// TIA Portal V17 export
// export: Created 2025-03-05T08:03:02.1046817Z, ExportSetting WithDefaults, DisplayName Totally Integrated Automation Portal, DisplayVersion V17 Update 8, DisplayName TIA Portal Openness, DisplayVersion V17 Update 8, DisplayName TIA Portal Version Control Interface, DisplayVersion V17, DisplayName SINAMICS Startdrive Advanced, DisplayVersion V17 SP2, DisplayName SINAMICS Startdrive G110M, G120, G120C, G120D, G120P, G115D, DisplayVersion V17 SP2, DisplayName SINAMICS Startdrive G130, G150, S120, S150, SINAMICS MV, S210, DisplayVersion V17 SP2, DisplayName STEP 7 Professional, DisplayVersion V17 Update 8, DisplayName SINUMERIK ONE STEP 7 Toolbox, DisplayVersion V17 Update 12, DisplayName SINUMERIK 840D sl STEP 7 Toolbox, DisplayVersion V17 Update 12, DisplayName STEP 7 Safety, DisplayVersion V17 Update 6, DisplayName WinCC Advanced, DisplayVersion V17 Update 8
FUNCTION "FC21013_POWDER_FEEDER_HOPPER" : Void   // FC21013, LAD
TITLE = FC21011 POWDER FEEDER HOPPER
{ S7_Optimized_Access := 'TRUE' }
VERSION : 0.1
// stored: AutoNumber false, IsIECCheckEnabled false, SetENOAutomatically false, UDAEnableTagReadback false
   VAR_TEMP
      AUX_PRESSURE : Int;
      AUX_DIGITAL1 : Bool;
      AUX_DIGITAL2 : Bool;
      AUX_SCATTER : Array[0..15] of Bool;
      PRESSURE_NORM : Real;
      PRESSURE_SCALE : Real;
      AUX_PRESSURE2 : Real;
      SCALED2 : Real;
   END_VAR
BEGIN

REGION Network 1: /////_UNIT_01_/////
END_REGION

REGION Network 2: CALL FB21013 POWDER FEEDER 1 HOPPER UNIT 01
   // 2#0000_0001 OPTIONS 0 BIT 0 LINE 1 ENABLED OPTION
   // 2#0000_0010 OPTIONS 0 BIT 1 LINE 2 ENABLED OPTION
   // 2#0000_0100 OPTIONS 0 BIT 2 SPARE
   // 2#0000_1000 OPTIONS 0 BIT 3 SPARE
   // 2#0001_0000 OPTIONS 0 BIT 4 SPARE
   // 2#0010_0000 OPTIONS 0 BIT 5 SPARE
   // 2#0100_0000 OPTIONS 0 BIT 6 SPARE
   // 2#1000_0000 OPTIONS 0 BIT 7 SPARE
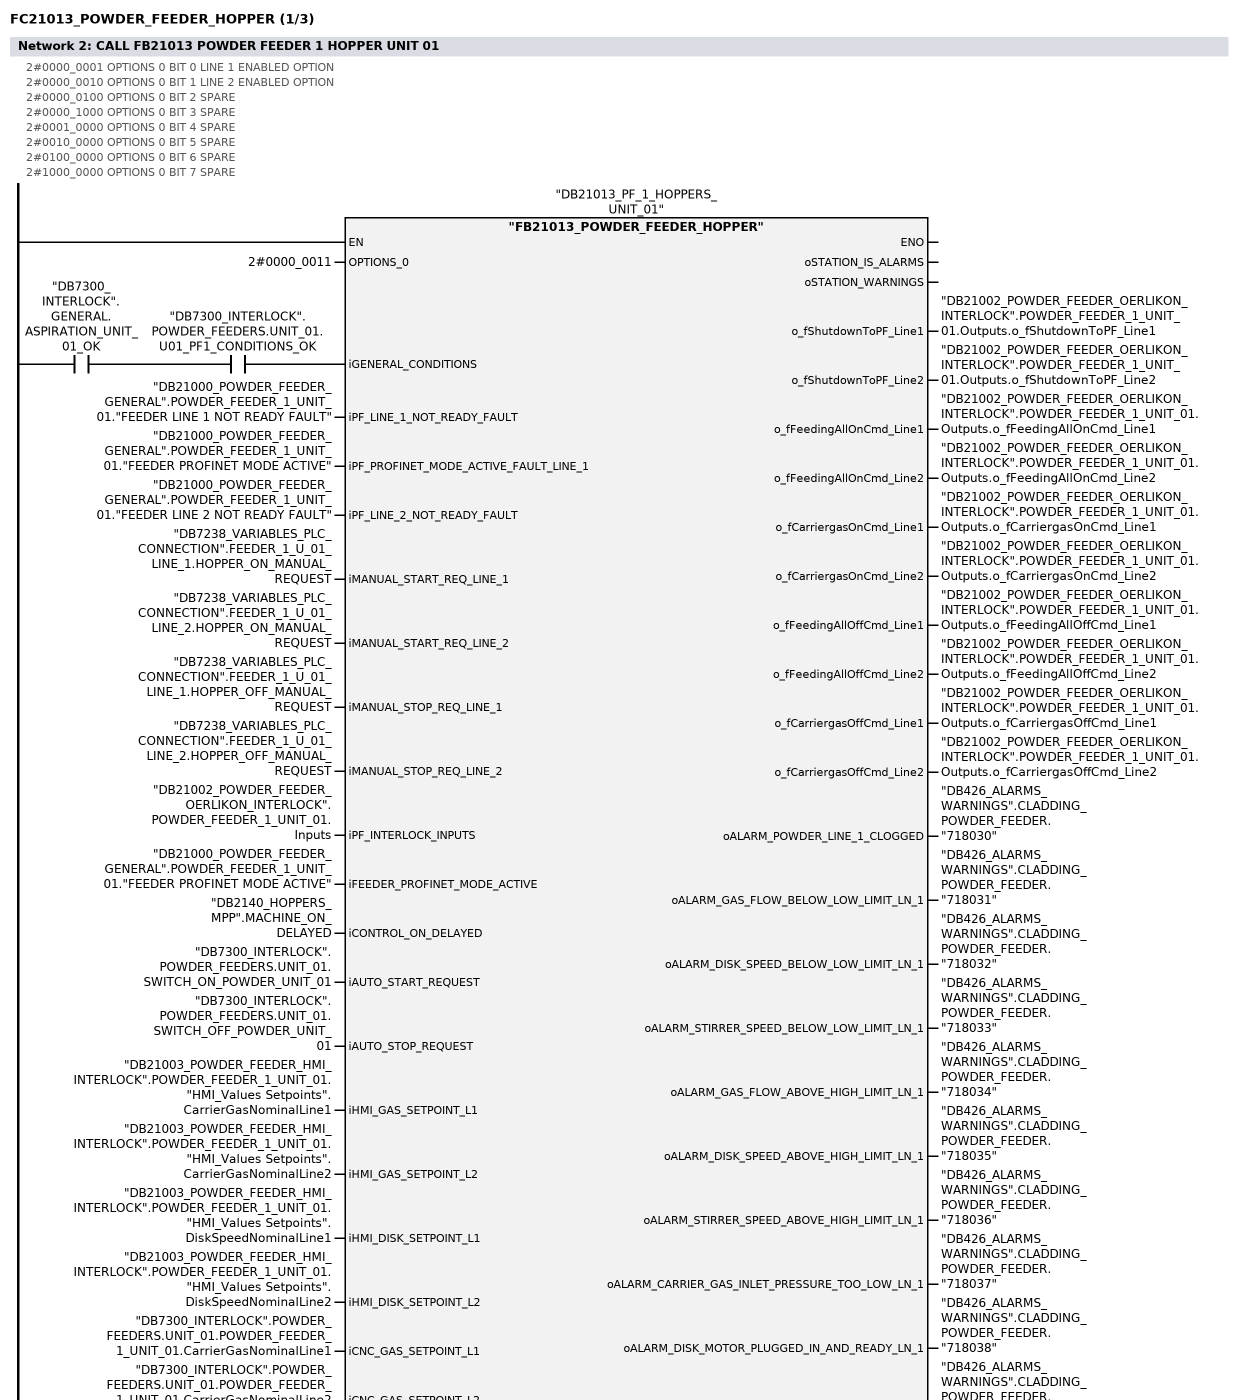
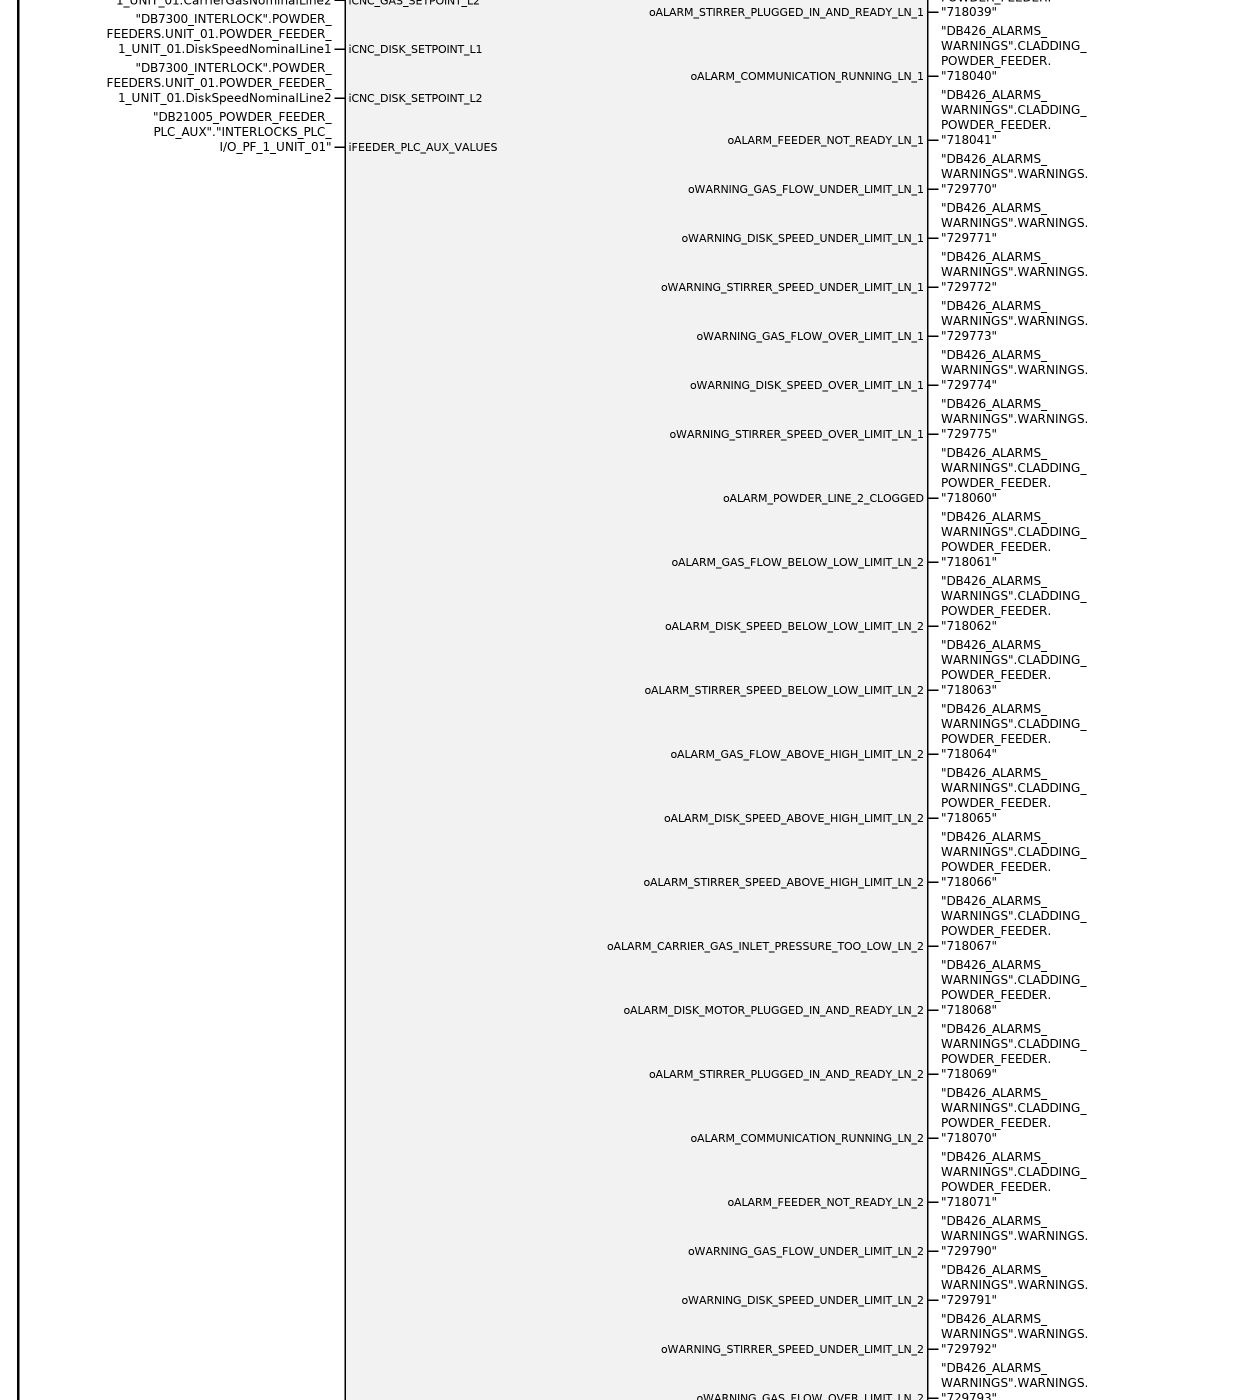
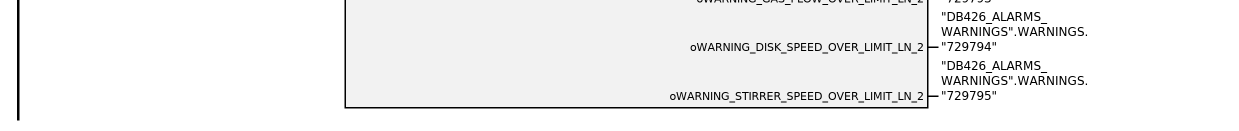
   RUNG wire#powerrail
      "DB21013_PF_1_HOPPERS_UNIT_01"(iGENERAL_CONDITIONS := wire#w1, OPTIONS_0 := 2#0000_0011, iPF_LINE_1_NOT_READY_FAULT := "DB21000_POWDER_FEEDER_GENERAL".POWDER_FEEDER_1_UNIT_01."FEEDER LINE 1 NOT READY FAULT", iPF_PROFINET_MODE_ACTIVE_FAULT_LINE_1 := "DB21000_POWDER_FEEDER_GENERAL".POWDER_FEEDER_1_UNIT_01."FEEDER PROFINET MODE ACTIVE", iPF_LINE_2_NOT_READY_FAULT := "DB21000_POWDER_FEEDER_GENERAL".POWDER_FEEDER_1_UNIT_01."FEEDER LINE 2 NOT READY FAULT", iMANUAL_START_REQ_LINE_1 := "DB7238_VARIABLES_PLC_CONNECTION".FEEDER_1_U_01_LINE_1.HOPPER_ON_MANUAL_REQUEST, iMANUAL_START_REQ_LINE_2 := "DB7238_VARIABLES_PLC_CONNECTION".FEEDER_1_U_01_LINE_2.HOPPER_ON_MANUAL_REQUEST, iMANUAL_STOP_REQ_LINE_1 := "DB7238_VARIABLES_PLC_CONNECTION".FEEDER_1_U_01_LINE_1.HOPPER_OFF_MANUAL_REQUEST, iMANUAL_STOP_REQ_LINE_2 := "DB7238_VARIABLES_PLC_CONNECTION".FEEDER_1_U_01_LINE_2.HOPPER_OFF_MANUAL_REQUEST, iPF_INTERLOCK_INPUTS := "DB21002_POWDER_FEEDER_OERLIKON_INTERLOCK".POWDER_FEEDER_1_UNIT_01.Inputs, iFEEDER_PROFINET_MODE_ACTIVE := "DB21000_POWDER_FEEDER_GENERAL".POWDER_FEEDER_1_UNIT_01."FEEDER PROFINET MODE ACTIVE", iCONTROL_ON_DELAYED := "DB2140_HOPPERS_MPP".MACHINE_ON_DELAYED, iAUTO_START_REQUEST := "DB7300_INTERLOCK".POWDER_FEEDERS.UNIT_01.SWITCH_ON_POWDER_UNIT_01, iAUTO_STOP_REQUEST := "DB7300_INTERLOCK".POWDER_FEEDERS.UNIT_01.SWITCH_OFF_POWDER_UNIT_01, iHMI_GAS_SETPOINT_L1 := "DB21003_POWDER_FEEDER_HMI_INTERLOCK".POWDER_FEEDER_1_UNIT_01."HMI_Values Setpoints".CarrierGasNominalLine1, iHMI_GAS_SETPOINT_L2 := "DB21003_POWDER_FEEDER_HMI_INTERLOCK".POWDER_FEEDER_1_UNIT_01."HMI_Values Setpoints".CarrierGasNominalLine2, iHMI_DISK_SETPOINT_L1 := "DB21003_POWDER_FEEDER_HMI_INTERLOCK".POWDER_FEEDER_1_UNIT_01."HMI_Values Setpoints".DiskSpeedNominalLine1, iHMI_DISK_SETPOINT_L2 := "DB21003_POWDER_FEEDER_HMI_INTERLOCK".POWDER_FEEDER_1_UNIT_01."HMI_Values Setpoints".DiskSpeedNominalLine2, iCNC_GAS_SETPOINT_L1 := "DB7300_INTERLOCK".POWDER_FEEDERS.UNIT_01.POWDER_FEEDER_1_UNIT_01.CarrierGasNominalLine1, iCNC_GAS_SETPOINT_L2 := "DB7300_INTERLOCK".POWDER_FEEDERS.UNIT_01.POWDER_FEEDER_1_UNIT_01.CarrierGasNominalLine2, iCNC_DISK_SETPOINT_L1 := "DB7300_INTERLOCK".POWDER_FEEDERS.UNIT_01.POWDER_FEEDER_1_UNIT_01.DiskSpeedNominalLine1, iCNC_DISK_SETPOINT_L2 := "DB7300_INTERLOCK".POWDER_FEEDERS.UNIT_01.POWDER_FEEDER_1_UNIT_01.DiskSpeedNominalLine2, iFEEDER_PLC_AUX_VALUES := "DB21005_POWDER_FEEDER_PLC_AUX"."INTERLOCKS_PLC_I/O_PF_1_UNIT_01", oSTATION_IS_ALARMS =>, oSTATION_WARNINGS =>, o_fShutdownToPF_Line1 => "DB21002_POWDER_FEEDER_OERLIKON_INTERLOCK".POWDER_FEEDER_1_UNIT_01.Outputs.o_fShutdownToPF_Line1, o_fShutdownToPF_Line2 => "DB21002_POWDER_FEEDER_OERLIKON_INTERLOCK".POWDER_FEEDER_1_UNIT_01.Outputs.o_fShutdownToPF_Line2, o_fFeedingAllOnCmd_Line1 => "DB21002_POWDER_FEEDER_OERLIKON_INTERLOCK".POWDER_FEEDER_1_UNIT_01.Outputs.o_fFeedingAllOnCmd_Line1, o_fFeedingAllOnCmd_Line2 => "DB21002_POWDER_FEEDER_OERLIKON_INTERLOCK".POWDER_FEEDER_1_UNIT_01.Outputs.o_fFeedingAllOnCmd_Line2, o_fCarriergasOnCmd_Line1 => "DB21002_POWDER_FEEDER_OERLIKON_INTERLOCK".POWDER_FEEDER_1_UNIT_01.Outputs.o_fCarriergasOnCmd_Line1, o_fCarriergasOnCmd_Line2 => "DB21002_POWDER_FEEDER_OERLIKON_INTERLOCK".POWDER_FEEDER_1_UNIT_01.Outputs.o_fCarriergasOnCmd_Line2, o_fFeedingAllOffCmd_Line1 => "DB21002_POWDER_FEEDER_OERLIKON_INTERLOCK".POWDER_FEEDER_1_UNIT_01.Outputs.o_fFeedingAllOffCmd_Line1, o_fFeedingAllOffCmd_Line2 => "DB21002_POWDER_FEEDER_OERLIKON_INTERLOCK".POWDER_FEEDER_1_UNIT_01.Outputs.o_fFeedingAllOffCmd_Line2, o_fCarriergasOffCmd_Line1 => "DB21002_POWDER_FEEDER_OERLIKON_INTERLOCK".POWDER_FEEDER_1_UNIT_01.Outputs.o_fCarriergasOffCmd_Line1, o_fCarriergasOffCmd_Line2 => "DB21002_POWDER_FEEDER_OERLIKON_INTERLOCK".POWDER_FEEDER_1_UNIT_01.Outputs.o_fCarriergasOffCmd_Line2, oALARM_POWDER_LINE_1_CLOGGED => "DB426_ALARMS_WARNINGS".CLADDING_POWDER_FEEDER."718030", oALARM_GAS_FLOW_BELOW_LOW_LIMIT_LN_1 => "DB426_ALARMS_WARNINGS".CLADDING_POWDER_FEEDER."718031", oALARM_DISK_SPEED_BELOW_LOW_LIMIT_LN_1 => "DB426_ALARMS_WARNINGS".CLADDING_POWDER_FEEDER."718032", oALARM_STIRRER_SPEED_BELOW_LOW_LIMIT_LN_1 => "DB426_ALARMS_WARNINGS".CLADDING_POWDER_FEEDER."718033", oALARM_GAS_FLOW_ABOVE_HIGH_LIMIT_LN_1 => "DB426_ALARMS_WARNINGS".CLADDING_POWDER_FEEDER."718034", oALARM_DISK_SPEED_ABOVE_HIGH_LIMIT_LN_1 => "DB426_ALARMS_WARNINGS".CLADDING_POWDER_FEEDER."718035", oALARM_STIRRER_SPEED_ABOVE_HIGH_LIMIT_LN_1 => "DB426_ALARMS_WARNINGS".CLADDING_POWDER_FEEDER."718036", oALARM_CARRIER_GAS_INLET_PRESSURE_TOO_LOW_LN_1 => "DB426_ALARMS_WARNINGS".CLADDING_POWDER_FEEDER."718037", oALARM_DISK_MOTOR_PLUGGED_IN_AND_READY_LN_1 => "DB426_ALARMS_WARNINGS".CLADDING_POWDER_FEEDER."718038", oALARM_STIRRER_PLUGGED_IN_AND_READY_LN_1 => "DB426_ALARMS_WARNINGS".CLADDING_POWDER_FEEDER."718039", oALARM_COMMUNICATION_RUNNING_LN_1 => "DB426_ALARMS_WARNINGS".CLADDING_POWDER_FEEDER."718040", oALARM_FEEDER_NOT_READY_LN_1 => "DB426_ALARMS_WARNINGS".CLADDING_POWDER_FEEDER."718041", oWARNING_GAS_FLOW_UNDER_LIMIT_LN_1 => "DB426_ALARMS_WARNINGS".WARNINGS."729770", oWARNING_DISK_SPEED_UNDER_LIMIT_LN_1 => "DB426_ALARMS_WARNINGS".WARNINGS."729771", oWARNING_STIRRER_SPEED_UNDER_LIMIT_LN_1 => "DB426_ALARMS_WARNINGS".WARNINGS."729772", oWARNING_GAS_FLOW_OVER_LIMIT_LN_1 => "DB426_ALARMS_WARNINGS".WARNINGS."729773", oWARNING_DISK_SPEED_OVER_LIMIT_LN_1 => "DB426_ALARMS_WARNINGS".WARNINGS."729774", oWARNING_STIRRER_SPEED_OVER_LIMIT_LN_1 => "DB426_ALARMS_WARNINGS".WARNINGS."729775", oALARM_POWDER_LINE_2_CLOGGED => "DB426_ALARMS_WARNINGS".CLADDING_POWDER_FEEDER."718060", oALARM_GAS_FLOW_BELOW_LOW_LIMIT_LN_2 => "DB426_ALARMS_WARNINGS".CLADDING_POWDER_FEEDER."718061", oALARM_DISK_SPEED_BELOW_LOW_LIMIT_LN_2 => "DB426_ALARMS_WARNINGS".CLADDING_POWDER_FEEDER."718062", oALARM_STIRRER_SPEED_BELOW_LOW_LIMIT_LN_2 => "DB426_ALARMS_WARNINGS".CLADDING_POWDER_FEEDER."718063", oALARM_GAS_FLOW_ABOVE_HIGH_LIMIT_LN_2 => "DB426_ALARMS_WARNINGS".CLADDING_POWDER_FEEDER."718064", oALARM_DISK_SPEED_ABOVE_HIGH_LIMIT_LN_2 => "DB426_ALARMS_WARNINGS".CLADDING_POWDER_FEEDER."718065", oALARM_STIRRER_SPEED_ABOVE_HIGH_LIMIT_LN_2 => "DB426_ALARMS_WARNINGS".CLADDING_POWDER_FEEDER."718066", oALARM_CARRIER_GAS_INLET_PRESSURE_TOO_LOW_LN_2 => "DB426_ALARMS_WARNINGS".CLADDING_POWDER_FEEDER."718067", oALARM_DISK_MOTOR_PLUGGED_IN_AND_READY_LN_2 => "DB426_ALARMS_WARNINGS".CLADDING_POWDER_FEEDER."718068", oALARM_STIRRER_PLUGGED_IN_AND_READY_LN_2 => "DB426_ALARMS_WARNINGS".CLADDING_POWDER_FEEDER."718069", oALARM_COMMUNICATION_RUNNING_LN_2 => "DB426_ALARMS_WARNINGS".CLADDING_POWDER_FEEDER."718070", oALARM_FEEDER_NOT_READY_LN_2 => "DB426_ALARMS_WARNINGS".CLADDING_POWDER_FEEDER."718071", oWARNING_GAS_FLOW_UNDER_LIMIT_LN_2 => "DB426_ALARMS_WARNINGS".WARNINGS."729790", oWARNING_DISK_SPEED_UNDER_LIMIT_LN_2 => "DB426_ALARMS_WARNINGS".WARNINGS."729791", oWARNING_STIRRER_SPEED_UNDER_LIMIT_LN_2 => "DB426_ALARMS_WARNINGS".WARNINGS."729792", oWARNING_GAS_FLOW_OVER_LIMIT_LN_2 => "DB426_ALARMS_WARNINGS".WARNINGS."729793", oWARNING_DISK_SPEED_OVER_LIMIT_LN_2 => "DB426_ALARMS_WARNINGS".WARNINGS."729794", oWARNING_STIRRER_SPEED_OVER_LIMIT_LN_2 => "DB426_ALARMS_WARNINGS".WARNINGS."729795")
   END_RUNG
   RUNG wire#powerrail
      Contact( "DB7300_INTERLOCK".GENERAL.ASPIRATION_UNIT_01_OK )
      Contact( "DB7300_INTERLOCK".POWDER_FEEDERS.UNIT_01.U01_PF1_CONDITIONS_OK )
   END_RUNG wire#w1
   // the same network as SCL:
   "DB21013_PF_1_HOPPERS_UNIT_01"(OPTIONS_0 := 2#0000_0011,   // "FB21013_POWDER_FEEDER_HOPPER"
                           iGENERAL_CONDITIONS := "DB7300_INTERLOCK".GENERAL.ASPIRATION_UNIT_01_OK AND "DB7300_INTERLOCK".POWDER_FEEDERS.UNIT_01.U01_PF1_CONDITIONS_OK,
                           iPF_LINE_1_NOT_READY_FAULT := "DB21000_POWDER_FEEDER_GENERAL".POWDER_FEEDER_1_UNIT_01."FEEDER LINE 1 NOT READY FAULT",
                           iPF_PROFINET_MODE_ACTIVE_FAULT_LINE_1 := "DB21000_POWDER_FEEDER_GENERAL".POWDER_FEEDER_1_UNIT_01."FEEDER PROFINET MODE ACTIVE",
                           iPF_LINE_2_NOT_READY_FAULT := "DB21000_POWDER_FEEDER_GENERAL".POWDER_FEEDER_1_UNIT_01."FEEDER LINE 2 NOT READY FAULT",
                           iMANUAL_START_REQ_LINE_1 := "DB7238_VARIABLES_PLC_CONNECTION".FEEDER_1_U_01_LINE_1.HOPPER_ON_MANUAL_REQUEST,
                           iMANUAL_START_REQ_LINE_2 := "DB7238_VARIABLES_PLC_CONNECTION".FEEDER_1_U_01_LINE_2.HOPPER_ON_MANUAL_REQUEST,
                           iMANUAL_STOP_REQ_LINE_1 := "DB7238_VARIABLES_PLC_CONNECTION".FEEDER_1_U_01_LINE_1.HOPPER_OFF_MANUAL_REQUEST,
                           iMANUAL_STOP_REQ_LINE_2 := "DB7238_VARIABLES_PLC_CONNECTION".FEEDER_1_U_01_LINE_2.HOPPER_OFF_MANUAL_REQUEST,
                           iPF_INTERLOCK_INPUTS := "DB21002_POWDER_FEEDER_OERLIKON_INTERLOCK".POWDER_FEEDER_1_UNIT_01.Inputs,
                           iFEEDER_PROFINET_MODE_ACTIVE := "DB21000_POWDER_FEEDER_GENERAL".POWDER_FEEDER_1_UNIT_01."FEEDER PROFINET MODE ACTIVE",
                           iCONTROL_ON_DELAYED := "DB2140_HOPPERS_MPP".MACHINE_ON_DELAYED,
                           iAUTO_START_REQUEST := "DB7300_INTERLOCK".POWDER_FEEDERS.UNIT_01.SWITCH_ON_POWDER_UNIT_01,
                           iAUTO_STOP_REQUEST := "DB7300_INTERLOCK".POWDER_FEEDERS.UNIT_01.SWITCH_OFF_POWDER_UNIT_01,
                           iHMI_GAS_SETPOINT_L1 := "DB21003_POWDER_FEEDER_HMI_INTERLOCK".POWDER_FEEDER_1_UNIT_01."HMI_Values Setpoints".CarrierGasNominalLine1,
                           iHMI_GAS_SETPOINT_L2 := "DB21003_POWDER_FEEDER_HMI_INTERLOCK".POWDER_FEEDER_1_UNIT_01."HMI_Values Setpoints".CarrierGasNominalLine2,
                           iHMI_DISK_SETPOINT_L1 := "DB21003_POWDER_FEEDER_HMI_INTERLOCK".POWDER_FEEDER_1_UNIT_01."HMI_Values Setpoints".DiskSpeedNominalLine1,
                           iHMI_DISK_SETPOINT_L2 := "DB21003_POWDER_FEEDER_HMI_INTERLOCK".POWDER_FEEDER_1_UNIT_01."HMI_Values Setpoints".DiskSpeedNominalLine2,
                           iCNC_GAS_SETPOINT_L1 := "DB7300_INTERLOCK".POWDER_FEEDERS.UNIT_01.POWDER_FEEDER_1_UNIT_01.CarrierGasNominalLine1,
                           iCNC_GAS_SETPOINT_L2 := "DB7300_INTERLOCK".POWDER_FEEDERS.UNIT_01.POWDER_FEEDER_1_UNIT_01.CarrierGasNominalLine2,
                           iCNC_DISK_SETPOINT_L1 := "DB7300_INTERLOCK".POWDER_FEEDERS.UNIT_01.POWDER_FEEDER_1_UNIT_01.DiskSpeedNominalLine1,
                           iCNC_DISK_SETPOINT_L2 := "DB7300_INTERLOCK".POWDER_FEEDERS.UNIT_01.POWDER_FEEDER_1_UNIT_01.DiskSpeedNominalLine2,
                           iFEEDER_PLC_AUX_VALUES := "DB21005_POWDER_FEEDER_PLC_AUX"."INTERLOCKS_PLC_I/O_PF_1_UNIT_01",
                           o_fShutdownToPF_Line1 => "DB21002_POWDER_FEEDER_OERLIKON_INTERLOCK".POWDER_FEEDER_1_UNIT_01.Outputs.o_fShutdownToPF_Line1,
                           o_fShutdownToPF_Line2 => "DB21002_POWDER_FEEDER_OERLIKON_INTERLOCK".POWDER_FEEDER_1_UNIT_01.Outputs.o_fShutdownToPF_Line2,
                           o_fFeedingAllOnCmd_Line1 => "DB21002_POWDER_FEEDER_OERLIKON_INTERLOCK".POWDER_FEEDER_1_UNIT_01.Outputs.o_fFeedingAllOnCmd_Line1,
                           o_fFeedingAllOnCmd_Line2 => "DB21002_POWDER_FEEDER_OERLIKON_INTERLOCK".POWDER_FEEDER_1_UNIT_01.Outputs.o_fFeedingAllOnCmd_Line2,
                           o_fCarriergasOnCmd_Line1 => "DB21002_POWDER_FEEDER_OERLIKON_INTERLOCK".POWDER_FEEDER_1_UNIT_01.Outputs.o_fCarriergasOnCmd_Line1,
                           o_fCarriergasOnCmd_Line2 => "DB21002_POWDER_FEEDER_OERLIKON_INTERLOCK".POWDER_FEEDER_1_UNIT_01.Outputs.o_fCarriergasOnCmd_Line2,
                           o_fFeedingAllOffCmd_Line1 => "DB21002_POWDER_FEEDER_OERLIKON_INTERLOCK".POWDER_FEEDER_1_UNIT_01.Outputs.o_fFeedingAllOffCmd_Line1,
                           o_fFeedingAllOffCmd_Line2 => "DB21002_POWDER_FEEDER_OERLIKON_INTERLOCK".POWDER_FEEDER_1_UNIT_01.Outputs.o_fFeedingAllOffCmd_Line2,
                           o_fCarriergasOffCmd_Line1 => "DB21002_POWDER_FEEDER_OERLIKON_INTERLOCK".POWDER_FEEDER_1_UNIT_01.Outputs.o_fCarriergasOffCmd_Line1,
                           o_fCarriergasOffCmd_Line2 => "DB21002_POWDER_FEEDER_OERLIKON_INTERLOCK".POWDER_FEEDER_1_UNIT_01.Outputs.o_fCarriergasOffCmd_Line2,
                           oALARM_POWDER_LINE_1_CLOGGED => "DB426_ALARMS_WARNINGS".CLADDING_POWDER_FEEDER."718030",
                           oALARM_GAS_FLOW_BELOW_LOW_LIMIT_LN_1 => "DB426_ALARMS_WARNINGS".CLADDING_POWDER_FEEDER."718031",
                           oALARM_DISK_SPEED_BELOW_LOW_LIMIT_LN_1 => "DB426_ALARMS_WARNINGS".CLADDING_POWDER_FEEDER."718032",
                           oALARM_STIRRER_SPEED_BELOW_LOW_LIMIT_LN_1 => "DB426_ALARMS_WARNINGS".CLADDING_POWDER_FEEDER."718033",
                           oALARM_GAS_FLOW_ABOVE_HIGH_LIMIT_LN_1 => "DB426_ALARMS_WARNINGS".CLADDING_POWDER_FEEDER."718034",
                           oALARM_DISK_SPEED_ABOVE_HIGH_LIMIT_LN_1 => "DB426_ALARMS_WARNINGS".CLADDING_POWDER_FEEDER."718035",
                           oALARM_STIRRER_SPEED_ABOVE_HIGH_LIMIT_LN_1 => "DB426_ALARMS_WARNINGS".CLADDING_POWDER_FEEDER."718036",
                           oALARM_CARRIER_GAS_INLET_PRESSURE_TOO_LOW_LN_1 => "DB426_ALARMS_WARNINGS".CLADDING_POWDER_FEEDER."718037",
                           oALARM_DISK_MOTOR_PLUGGED_IN_AND_READY_LN_1 => "DB426_ALARMS_WARNINGS".CLADDING_POWDER_FEEDER."718038",
                           oALARM_STIRRER_PLUGGED_IN_AND_READY_LN_1 => "DB426_ALARMS_WARNINGS".CLADDING_POWDER_FEEDER."718039",
                           oALARM_COMMUNICATION_RUNNING_LN_1 => "DB426_ALARMS_WARNINGS".CLADDING_POWDER_FEEDER."718040",
                           oALARM_FEEDER_NOT_READY_LN_1 => "DB426_ALARMS_WARNINGS".CLADDING_POWDER_FEEDER."718041",
                           oWARNING_GAS_FLOW_UNDER_LIMIT_LN_1 => "DB426_ALARMS_WARNINGS".WARNINGS."729770",
                           oWARNING_DISK_SPEED_UNDER_LIMIT_LN_1 => "DB426_ALARMS_WARNINGS".WARNINGS."729771",
                           oWARNING_STIRRER_SPEED_UNDER_LIMIT_LN_1 => "DB426_ALARMS_WARNINGS".WARNINGS."729772",
                           oWARNING_GAS_FLOW_OVER_LIMIT_LN_1 => "DB426_ALARMS_WARNINGS".WARNINGS."729773",
                           oWARNING_DISK_SPEED_OVER_LIMIT_LN_1 => "DB426_ALARMS_WARNINGS".WARNINGS."729774",
                           oWARNING_STIRRER_SPEED_OVER_LIMIT_LN_1 => "DB426_ALARMS_WARNINGS".WARNINGS."729775",
                           oALARM_POWDER_LINE_2_CLOGGED => "DB426_ALARMS_WARNINGS".CLADDING_POWDER_FEEDER."718060",
                           oALARM_GAS_FLOW_BELOW_LOW_LIMIT_LN_2 => "DB426_ALARMS_WARNINGS".CLADDING_POWDER_FEEDER."718061",
                           oALARM_DISK_SPEED_BELOW_LOW_LIMIT_LN_2 => "DB426_ALARMS_WARNINGS".CLADDING_POWDER_FEEDER."718062",
                           oALARM_STIRRER_SPEED_BELOW_LOW_LIMIT_LN_2 => "DB426_ALARMS_WARNINGS".CLADDING_POWDER_FEEDER."718063",
                           oALARM_GAS_FLOW_ABOVE_HIGH_LIMIT_LN_2 => "DB426_ALARMS_WARNINGS".CLADDING_POWDER_FEEDER."718064",
                           oALARM_DISK_SPEED_ABOVE_HIGH_LIMIT_LN_2 => "DB426_ALARMS_WARNINGS".CLADDING_POWDER_FEEDER."718065",
                           oALARM_STIRRER_SPEED_ABOVE_HIGH_LIMIT_LN_2 => "DB426_ALARMS_WARNINGS".CLADDING_POWDER_FEEDER."718066",
                           oALARM_CARRIER_GAS_INLET_PRESSURE_TOO_LOW_LN_2 => "DB426_ALARMS_WARNINGS".CLADDING_POWDER_FEEDER."718067",
                           oALARM_DISK_MOTOR_PLUGGED_IN_AND_READY_LN_2 => "DB426_ALARMS_WARNINGS".CLADDING_POWDER_FEEDER."718068",
                           oALARM_STIRRER_PLUGGED_IN_AND_READY_LN_2 => "DB426_ALARMS_WARNINGS".CLADDING_POWDER_FEEDER."718069",
                           oALARM_COMMUNICATION_RUNNING_LN_2 => "DB426_ALARMS_WARNINGS".CLADDING_POWDER_FEEDER."718070",
                           oALARM_FEEDER_NOT_READY_LN_2 => "DB426_ALARMS_WARNINGS".CLADDING_POWDER_FEEDER."718071",
                           oWARNING_GAS_FLOW_UNDER_LIMIT_LN_2 => "DB426_ALARMS_WARNINGS".WARNINGS."729790",
                           oWARNING_DISK_SPEED_UNDER_LIMIT_LN_2 => "DB426_ALARMS_WARNINGS".WARNINGS."729791",
                           oWARNING_STIRRER_SPEED_UNDER_LIMIT_LN_2 => "DB426_ALARMS_WARNINGS".WARNINGS."729792",
                           oWARNING_GAS_FLOW_OVER_LIMIT_LN_2 => "DB426_ALARMS_WARNINGS".WARNINGS."729793",
                           oWARNING_DISK_SPEED_OVER_LIMIT_LN_2 => "DB426_ALARMS_WARNINGS".WARNINGS."729794",
                           oWARNING_STIRRER_SPEED_OVER_LIMIT_LN_2 => "DB426_ALARMS_WARNINGS".WARNINGS."729795");
END_REGION

REGION Network 3: /////_UNIT_02_/////
END_REGION

REGION Network 4: CALL FB21013 POWDER FEEDER 1 HOPPER UNIT 02
   // 2#0000_0001 OPTIONS 0 BIT 0 LINE 1 ENABLED OPTION
   // 2#0000_0010 OPTIONS 0 BIT 1 LINE 2 ENABLED OPTION
   // 2#0000_0100 OPTIONS 0 BIT 2 SPARE
   // 2#0000_1000 OPTIONS 0 BIT 3 SPARE
   // 2#0001_0000 OPTIONS 0 BIT 4 SPARE
   // 2#0010_0000 OPTIONS 0 BIT 5 SPARE
   // 2#0100_0000 OPTIONS 0 BIT 6 SPARE
   // 2#1000_0000 OPTIONS 0 BIT 7 SPARE
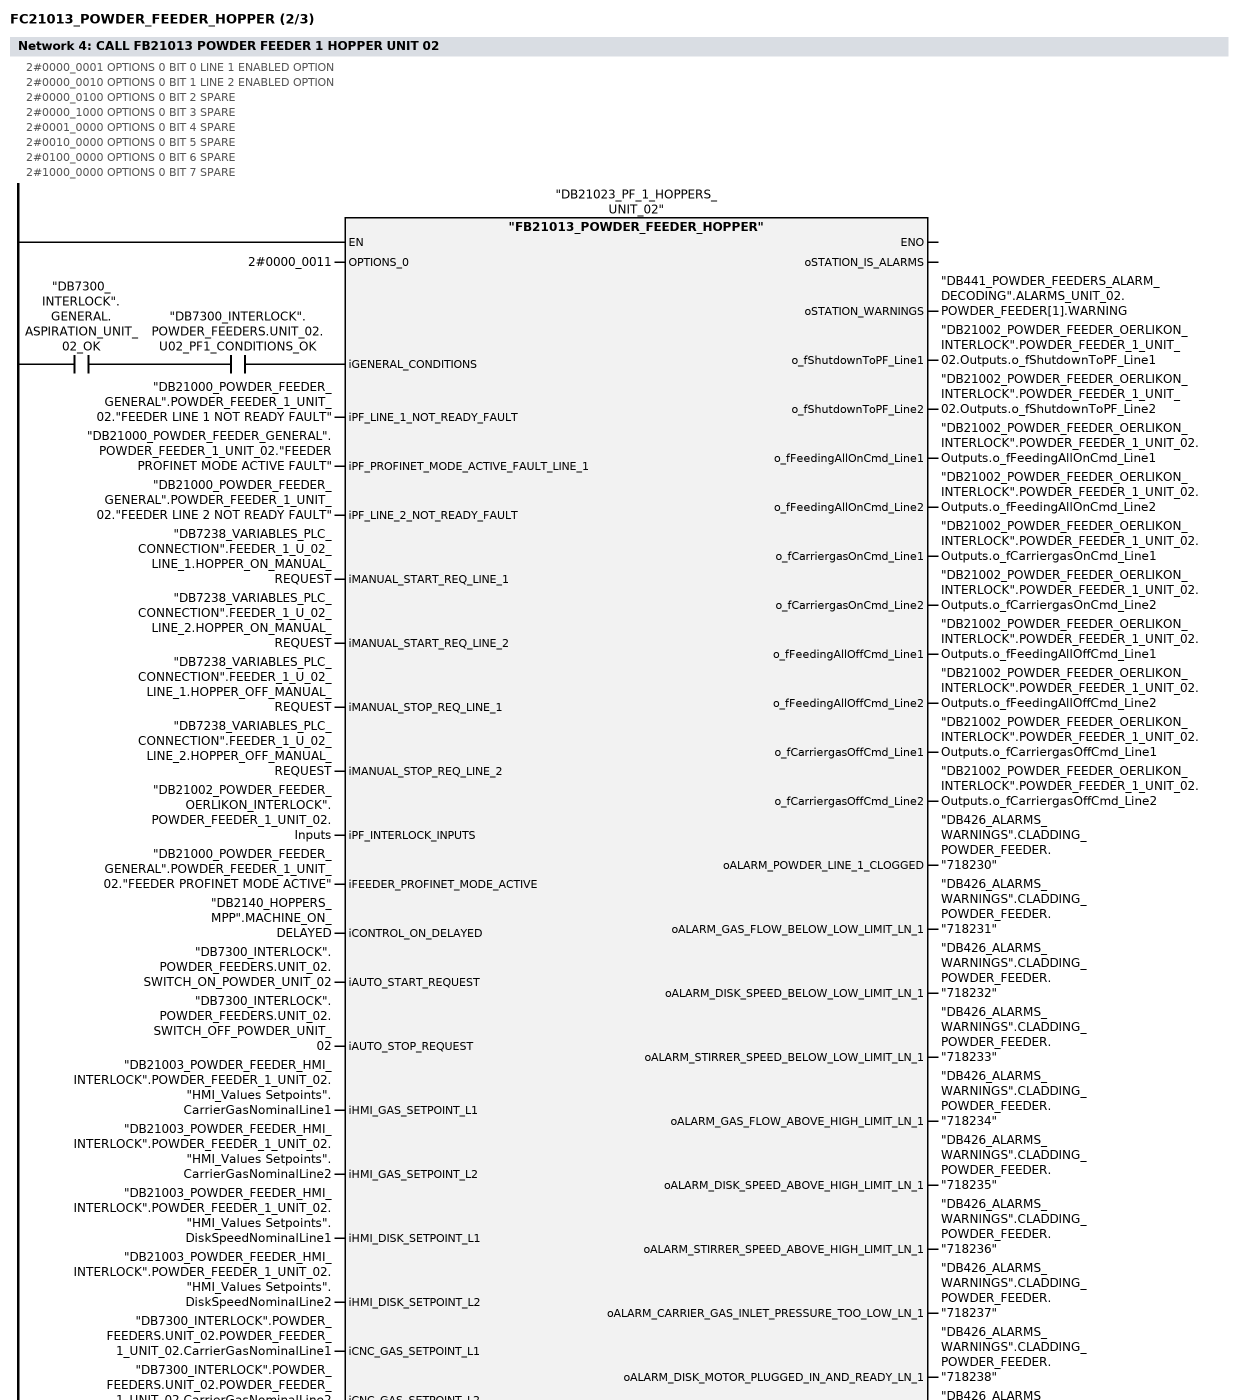
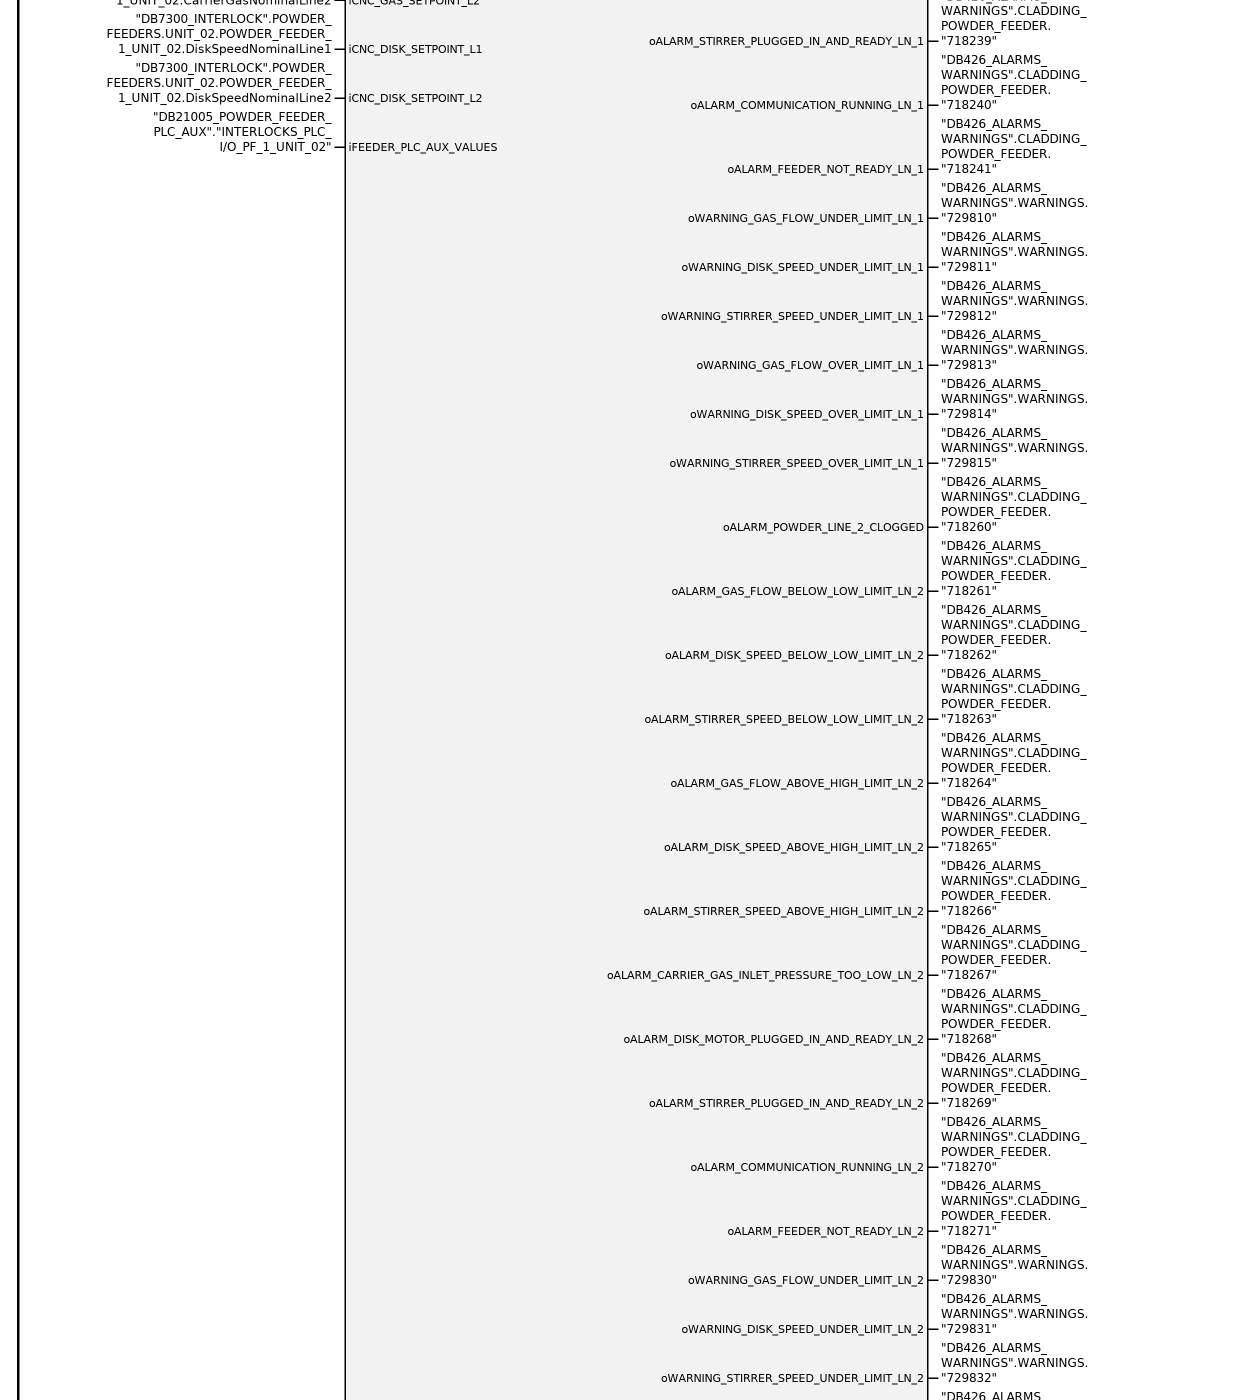
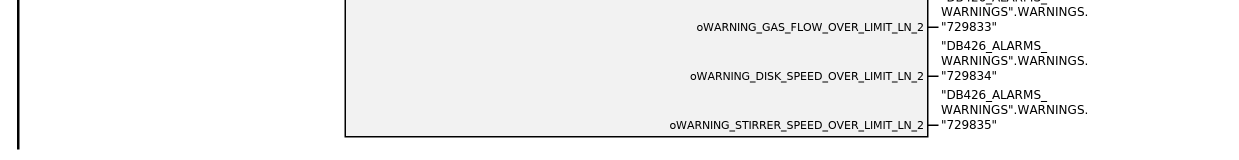
   RUNG wire#powerrail
      "DB21023_PF_1_HOPPERS_UNIT_02"(iGENERAL_CONDITIONS := wire#w1, OPTIONS_0 := 2#0000_0011, iPF_LINE_1_NOT_READY_FAULT := "DB21000_POWDER_FEEDER_GENERAL".POWDER_FEEDER_1_UNIT_02."FEEDER LINE 1 NOT READY FAULT", iPF_PROFINET_MODE_ACTIVE_FAULT_LINE_1 := "DB21000_POWDER_FEEDER_GENERAL".POWDER_FEEDER_1_UNIT_02."FEEDER PROFINET MODE ACTIVE FAULT", iPF_LINE_2_NOT_READY_FAULT := "DB21000_POWDER_FEEDER_GENERAL".POWDER_FEEDER_1_UNIT_02."FEEDER LINE 2 NOT READY FAULT", iMANUAL_START_REQ_LINE_1 := "DB7238_VARIABLES_PLC_CONNECTION".FEEDER_1_U_02_LINE_1.HOPPER_ON_MANUAL_REQUEST, iMANUAL_START_REQ_LINE_2 := "DB7238_VARIABLES_PLC_CONNECTION".FEEDER_1_U_02_LINE_2.HOPPER_ON_MANUAL_REQUEST, iMANUAL_STOP_REQ_LINE_1 := "DB7238_VARIABLES_PLC_CONNECTION".FEEDER_1_U_02_LINE_1.HOPPER_OFF_MANUAL_REQUEST, iMANUAL_STOP_REQ_LINE_2 := "DB7238_VARIABLES_PLC_CONNECTION".FEEDER_1_U_02_LINE_2.HOPPER_OFF_MANUAL_REQUEST, iPF_INTERLOCK_INPUTS := "DB21002_POWDER_FEEDER_OERLIKON_INTERLOCK".POWDER_FEEDER_1_UNIT_02.Inputs, iFEEDER_PROFINET_MODE_ACTIVE := "DB21000_POWDER_FEEDER_GENERAL".POWDER_FEEDER_1_UNIT_02."FEEDER PROFINET MODE ACTIVE", iCONTROL_ON_DELAYED := "DB2140_HOPPERS_MPP".MACHINE_ON_DELAYED, iAUTO_START_REQUEST := "DB7300_INTERLOCK".POWDER_FEEDERS.UNIT_02.SWITCH_ON_POWDER_UNIT_02, iAUTO_STOP_REQUEST := "DB7300_INTERLOCK".POWDER_FEEDERS.UNIT_02.SWITCH_OFF_POWDER_UNIT_02, iHMI_GAS_SETPOINT_L1 := "DB21003_POWDER_FEEDER_HMI_INTERLOCK".POWDER_FEEDER_1_UNIT_02."HMI_Values Setpoints".CarrierGasNominalLine1, iHMI_GAS_SETPOINT_L2 := "DB21003_POWDER_FEEDER_HMI_INTERLOCK".POWDER_FEEDER_1_UNIT_02."HMI_Values Setpoints".CarrierGasNominalLine2, iHMI_DISK_SETPOINT_L1 := "DB21003_POWDER_FEEDER_HMI_INTERLOCK".POWDER_FEEDER_1_UNIT_02."HMI_Values Setpoints".DiskSpeedNominalLine1, iHMI_DISK_SETPOINT_L2 := "DB21003_POWDER_FEEDER_HMI_INTERLOCK".POWDER_FEEDER_1_UNIT_02."HMI_Values Setpoints".DiskSpeedNominalLine2, iCNC_GAS_SETPOINT_L1 := "DB7300_INTERLOCK".POWDER_FEEDERS.UNIT_02.POWDER_FEEDER_1_UNIT_02.CarrierGasNominalLine1, iCNC_GAS_SETPOINT_L2 := "DB7300_INTERLOCK".POWDER_FEEDERS.UNIT_02.POWDER_FEEDER_1_UNIT_02.CarrierGasNominalLine2, iCNC_DISK_SETPOINT_L1 := "DB7300_INTERLOCK".POWDER_FEEDERS.UNIT_02.POWDER_FEEDER_1_UNIT_02.DiskSpeedNominalLine1, iCNC_DISK_SETPOINT_L2 := "DB7300_INTERLOCK".POWDER_FEEDERS.UNIT_02.POWDER_FEEDER_1_UNIT_02.DiskSpeedNominalLine2, iFEEDER_PLC_AUX_VALUES := "DB21005_POWDER_FEEDER_PLC_AUX"."INTERLOCKS_PLC_I/O_PF_1_UNIT_02", oSTATION_IS_ALARMS =>, oSTATION_WARNINGS => "DB441_POWDER_FEEDERS_ALARM_DECODING".ALARMS_UNIT_02.POWDER_FEEDER[1].WARNING, o_fShutdownToPF_Line1 => "DB21002_POWDER_FEEDER_OERLIKON_INTERLOCK".POWDER_FEEDER_1_UNIT_02.Outputs.o_fShutdownToPF_Line1, o_fShutdownToPF_Line2 => "DB21002_POWDER_FEEDER_OERLIKON_INTERLOCK".POWDER_FEEDER_1_UNIT_02.Outputs.o_fShutdownToPF_Line2, o_fFeedingAllOnCmd_Line1 => "DB21002_POWDER_FEEDER_OERLIKON_INTERLOCK".POWDER_FEEDER_1_UNIT_02.Outputs.o_fFeedingAllOnCmd_Line1, o_fFeedingAllOnCmd_Line2 => "DB21002_POWDER_FEEDER_OERLIKON_INTERLOCK".POWDER_FEEDER_1_UNIT_02.Outputs.o_fFeedingAllOnCmd_Line2, o_fCarriergasOnCmd_Line1 => "DB21002_POWDER_FEEDER_OERLIKON_INTERLOCK".POWDER_FEEDER_1_UNIT_02.Outputs.o_fCarriergasOnCmd_Line1, o_fCarriergasOnCmd_Line2 => "DB21002_POWDER_FEEDER_OERLIKON_INTERLOCK".POWDER_FEEDER_1_UNIT_02.Outputs.o_fCarriergasOnCmd_Line2, o_fFeedingAllOffCmd_Line1 => "DB21002_POWDER_FEEDER_OERLIKON_INTERLOCK".POWDER_FEEDER_1_UNIT_02.Outputs.o_fFeedingAllOffCmd_Line1, o_fFeedingAllOffCmd_Line2 => "DB21002_POWDER_FEEDER_OERLIKON_INTERLOCK".POWDER_FEEDER_1_UNIT_02.Outputs.o_fFeedingAllOffCmd_Line2, o_fCarriergasOffCmd_Line1 => "DB21002_POWDER_FEEDER_OERLIKON_INTERLOCK".POWDER_FEEDER_1_UNIT_02.Outputs.o_fCarriergasOffCmd_Line1, o_fCarriergasOffCmd_Line2 => "DB21002_POWDER_FEEDER_OERLIKON_INTERLOCK".POWDER_FEEDER_1_UNIT_02.Outputs.o_fCarriergasOffCmd_Line2, oALARM_POWDER_LINE_1_CLOGGED => "DB426_ALARMS_WARNINGS".CLADDING_POWDER_FEEDER."718230", oALARM_GAS_FLOW_BELOW_LOW_LIMIT_LN_1 => "DB426_ALARMS_WARNINGS".CLADDING_POWDER_FEEDER."718231", oALARM_DISK_SPEED_BELOW_LOW_LIMIT_LN_1 => "DB426_ALARMS_WARNINGS".CLADDING_POWDER_FEEDER."718232", oALARM_STIRRER_SPEED_BELOW_LOW_LIMIT_LN_1 => "DB426_ALARMS_WARNINGS".CLADDING_POWDER_FEEDER."718233", oALARM_GAS_FLOW_ABOVE_HIGH_LIMIT_LN_1 => "DB426_ALARMS_WARNINGS".CLADDING_POWDER_FEEDER."718234", oALARM_DISK_SPEED_ABOVE_HIGH_LIMIT_LN_1 => "DB426_ALARMS_WARNINGS".CLADDING_POWDER_FEEDER."718235", oALARM_STIRRER_SPEED_ABOVE_HIGH_LIMIT_LN_1 => "DB426_ALARMS_WARNINGS".CLADDING_POWDER_FEEDER."718236", oALARM_CARRIER_GAS_INLET_PRESSURE_TOO_LOW_LN_1 => "DB426_ALARMS_WARNINGS".CLADDING_POWDER_FEEDER."718237", oALARM_DISK_MOTOR_PLUGGED_IN_AND_READY_LN_1 => "DB426_ALARMS_WARNINGS".CLADDING_POWDER_FEEDER."718238", oALARM_STIRRER_PLUGGED_IN_AND_READY_LN_1 => "DB426_ALARMS_WARNINGS".CLADDING_POWDER_FEEDER."718239", oALARM_COMMUNICATION_RUNNING_LN_1 => "DB426_ALARMS_WARNINGS".CLADDING_POWDER_FEEDER."718240", oALARM_FEEDER_NOT_READY_LN_1 => "DB426_ALARMS_WARNINGS".CLADDING_POWDER_FEEDER."718241", oWARNING_GAS_FLOW_UNDER_LIMIT_LN_1 => "DB426_ALARMS_WARNINGS".WARNINGS."729810", oWARNING_DISK_SPEED_UNDER_LIMIT_LN_1 => "DB426_ALARMS_WARNINGS".WARNINGS."729811", oWARNING_STIRRER_SPEED_UNDER_LIMIT_LN_1 => "DB426_ALARMS_WARNINGS".WARNINGS."729812", oWARNING_GAS_FLOW_OVER_LIMIT_LN_1 => "DB426_ALARMS_WARNINGS".WARNINGS."729813", oWARNING_DISK_SPEED_OVER_LIMIT_LN_1 => "DB426_ALARMS_WARNINGS".WARNINGS."729814", oWARNING_STIRRER_SPEED_OVER_LIMIT_LN_1 => "DB426_ALARMS_WARNINGS".WARNINGS."729815", oALARM_POWDER_LINE_2_CLOGGED => "DB426_ALARMS_WARNINGS".CLADDING_POWDER_FEEDER."718260", oALARM_GAS_FLOW_BELOW_LOW_LIMIT_LN_2 => "DB426_ALARMS_WARNINGS".CLADDING_POWDER_FEEDER."718261", oALARM_DISK_SPEED_BELOW_LOW_LIMIT_LN_2 => "DB426_ALARMS_WARNINGS".CLADDING_POWDER_FEEDER."718262", oALARM_STIRRER_SPEED_BELOW_LOW_LIMIT_LN_2 => "DB426_ALARMS_WARNINGS".CLADDING_POWDER_FEEDER."718263", oALARM_GAS_FLOW_ABOVE_HIGH_LIMIT_LN_2 => "DB426_ALARMS_WARNINGS".CLADDING_POWDER_FEEDER."718264", oALARM_DISK_SPEED_ABOVE_HIGH_LIMIT_LN_2 => "DB426_ALARMS_WARNINGS".CLADDING_POWDER_FEEDER."718265", oALARM_STIRRER_SPEED_ABOVE_HIGH_LIMIT_LN_2 => "DB426_ALARMS_WARNINGS".CLADDING_POWDER_FEEDER."718266", oALARM_CARRIER_GAS_INLET_PRESSURE_TOO_LOW_LN_2 => "DB426_ALARMS_WARNINGS".CLADDING_POWDER_FEEDER."718267", oALARM_DISK_MOTOR_PLUGGED_IN_AND_READY_LN_2 => "DB426_ALARMS_WARNINGS".CLADDING_POWDER_FEEDER."718268", oALARM_STIRRER_PLUGGED_IN_AND_READY_LN_2 => "DB426_ALARMS_WARNINGS".CLADDING_POWDER_FEEDER."718269", oALARM_COMMUNICATION_RUNNING_LN_2 => "DB426_ALARMS_WARNINGS".CLADDING_POWDER_FEEDER."718270", oALARM_FEEDER_NOT_READY_LN_2 => "DB426_ALARMS_WARNINGS".CLADDING_POWDER_FEEDER."718271", oWARNING_GAS_FLOW_UNDER_LIMIT_LN_2 => "DB426_ALARMS_WARNINGS".WARNINGS."729830", oWARNING_DISK_SPEED_UNDER_LIMIT_LN_2 => "DB426_ALARMS_WARNINGS".WARNINGS."729831", oWARNING_STIRRER_SPEED_UNDER_LIMIT_LN_2 => "DB426_ALARMS_WARNINGS".WARNINGS."729832", oWARNING_GAS_FLOW_OVER_LIMIT_LN_2 => "DB426_ALARMS_WARNINGS".WARNINGS."729833", oWARNING_DISK_SPEED_OVER_LIMIT_LN_2 => "DB426_ALARMS_WARNINGS".WARNINGS."729834", oWARNING_STIRRER_SPEED_OVER_LIMIT_LN_2 => "DB426_ALARMS_WARNINGS".WARNINGS."729835")
   END_RUNG
   RUNG wire#powerrail
      Contact( "DB7300_INTERLOCK".GENERAL.ASPIRATION_UNIT_02_OK )
      Contact( "DB7300_INTERLOCK".POWDER_FEEDERS.UNIT_02.U02_PF1_CONDITIONS_OK )
   END_RUNG wire#w1
   // the same network as SCL:
   "DB21023_PF_1_HOPPERS_UNIT_02"(OPTIONS_0 := 2#0000_0011,   // "FB21013_POWDER_FEEDER_HOPPER"
                           iGENERAL_CONDITIONS := "DB7300_INTERLOCK".GENERAL.ASPIRATION_UNIT_02_OK AND "DB7300_INTERLOCK".POWDER_FEEDERS.UNIT_02.U02_PF1_CONDITIONS_OK,
                           iPF_LINE_1_NOT_READY_FAULT := "DB21000_POWDER_FEEDER_GENERAL".POWDER_FEEDER_1_UNIT_02."FEEDER LINE 1 NOT READY FAULT",
                           iPF_PROFINET_MODE_ACTIVE_FAULT_LINE_1 := "DB21000_POWDER_FEEDER_GENERAL".POWDER_FEEDER_1_UNIT_02."FEEDER PROFINET MODE ACTIVE FAULT",
                           iPF_LINE_2_NOT_READY_FAULT := "DB21000_POWDER_FEEDER_GENERAL".POWDER_FEEDER_1_UNIT_02."FEEDER LINE 2 NOT READY FAULT",
                           iMANUAL_START_REQ_LINE_1 := "DB7238_VARIABLES_PLC_CONNECTION".FEEDER_1_U_02_LINE_1.HOPPER_ON_MANUAL_REQUEST,
                           iMANUAL_START_REQ_LINE_2 := "DB7238_VARIABLES_PLC_CONNECTION".FEEDER_1_U_02_LINE_2.HOPPER_ON_MANUAL_REQUEST,
                           iMANUAL_STOP_REQ_LINE_1 := "DB7238_VARIABLES_PLC_CONNECTION".FEEDER_1_U_02_LINE_1.HOPPER_OFF_MANUAL_REQUEST,
                           iMANUAL_STOP_REQ_LINE_2 := "DB7238_VARIABLES_PLC_CONNECTION".FEEDER_1_U_02_LINE_2.HOPPER_OFF_MANUAL_REQUEST,
                           iPF_INTERLOCK_INPUTS := "DB21002_POWDER_FEEDER_OERLIKON_INTERLOCK".POWDER_FEEDER_1_UNIT_02.Inputs,
                           iFEEDER_PROFINET_MODE_ACTIVE := "DB21000_POWDER_FEEDER_GENERAL".POWDER_FEEDER_1_UNIT_02."FEEDER PROFINET MODE ACTIVE",
                           iCONTROL_ON_DELAYED := "DB2140_HOPPERS_MPP".MACHINE_ON_DELAYED,
                           iAUTO_START_REQUEST := "DB7300_INTERLOCK".POWDER_FEEDERS.UNIT_02.SWITCH_ON_POWDER_UNIT_02,
                           iAUTO_STOP_REQUEST := "DB7300_INTERLOCK".POWDER_FEEDERS.UNIT_02.SWITCH_OFF_POWDER_UNIT_02,
                           iHMI_GAS_SETPOINT_L1 := "DB21003_POWDER_FEEDER_HMI_INTERLOCK".POWDER_FEEDER_1_UNIT_02."HMI_Values Setpoints".CarrierGasNominalLine1,
                           iHMI_GAS_SETPOINT_L2 := "DB21003_POWDER_FEEDER_HMI_INTERLOCK".POWDER_FEEDER_1_UNIT_02."HMI_Values Setpoints".CarrierGasNominalLine2,
                           iHMI_DISK_SETPOINT_L1 := "DB21003_POWDER_FEEDER_HMI_INTERLOCK".POWDER_FEEDER_1_UNIT_02."HMI_Values Setpoints".DiskSpeedNominalLine1,
                           iHMI_DISK_SETPOINT_L2 := "DB21003_POWDER_FEEDER_HMI_INTERLOCK".POWDER_FEEDER_1_UNIT_02."HMI_Values Setpoints".DiskSpeedNominalLine2,
                           iCNC_GAS_SETPOINT_L1 := "DB7300_INTERLOCK".POWDER_FEEDERS.UNIT_02.POWDER_FEEDER_1_UNIT_02.CarrierGasNominalLine1,
                           iCNC_GAS_SETPOINT_L2 := "DB7300_INTERLOCK".POWDER_FEEDERS.UNIT_02.POWDER_FEEDER_1_UNIT_02.CarrierGasNominalLine2,
                           iCNC_DISK_SETPOINT_L1 := "DB7300_INTERLOCK".POWDER_FEEDERS.UNIT_02.POWDER_FEEDER_1_UNIT_02.DiskSpeedNominalLine1,
                           iCNC_DISK_SETPOINT_L2 := "DB7300_INTERLOCK".POWDER_FEEDERS.UNIT_02.POWDER_FEEDER_1_UNIT_02.DiskSpeedNominalLine2,
                           iFEEDER_PLC_AUX_VALUES := "DB21005_POWDER_FEEDER_PLC_AUX"."INTERLOCKS_PLC_I/O_PF_1_UNIT_02",
                           oSTATION_WARNINGS => "DB441_POWDER_FEEDERS_ALARM_DECODING".ALARMS_UNIT_02.POWDER_FEEDER[1].WARNING,
                           o_fShutdownToPF_Line1 => "DB21002_POWDER_FEEDER_OERLIKON_INTERLOCK".POWDER_FEEDER_1_UNIT_02.Outputs.o_fShutdownToPF_Line1,
                           o_fShutdownToPF_Line2 => "DB21002_POWDER_FEEDER_OERLIKON_INTERLOCK".POWDER_FEEDER_1_UNIT_02.Outputs.o_fShutdownToPF_Line2,
                           o_fFeedingAllOnCmd_Line1 => "DB21002_POWDER_FEEDER_OERLIKON_INTERLOCK".POWDER_FEEDER_1_UNIT_02.Outputs.o_fFeedingAllOnCmd_Line1,
                           o_fFeedingAllOnCmd_Line2 => "DB21002_POWDER_FEEDER_OERLIKON_INTERLOCK".POWDER_FEEDER_1_UNIT_02.Outputs.o_fFeedingAllOnCmd_Line2,
                           o_fCarriergasOnCmd_Line1 => "DB21002_POWDER_FEEDER_OERLIKON_INTERLOCK".POWDER_FEEDER_1_UNIT_02.Outputs.o_fCarriergasOnCmd_Line1,
                           o_fCarriergasOnCmd_Line2 => "DB21002_POWDER_FEEDER_OERLIKON_INTERLOCK".POWDER_FEEDER_1_UNIT_02.Outputs.o_fCarriergasOnCmd_Line2,
                           o_fFeedingAllOffCmd_Line1 => "DB21002_POWDER_FEEDER_OERLIKON_INTERLOCK".POWDER_FEEDER_1_UNIT_02.Outputs.o_fFeedingAllOffCmd_Line1,
                           o_fFeedingAllOffCmd_Line2 => "DB21002_POWDER_FEEDER_OERLIKON_INTERLOCK".POWDER_FEEDER_1_UNIT_02.Outputs.o_fFeedingAllOffCmd_Line2,
                           o_fCarriergasOffCmd_Line1 => "DB21002_POWDER_FEEDER_OERLIKON_INTERLOCK".POWDER_FEEDER_1_UNIT_02.Outputs.o_fCarriergasOffCmd_Line1,
                           o_fCarriergasOffCmd_Line2 => "DB21002_POWDER_FEEDER_OERLIKON_INTERLOCK".POWDER_FEEDER_1_UNIT_02.Outputs.o_fCarriergasOffCmd_Line2,
                           oALARM_POWDER_LINE_1_CLOGGED => "DB426_ALARMS_WARNINGS".CLADDING_POWDER_FEEDER."718230",
                           oALARM_GAS_FLOW_BELOW_LOW_LIMIT_LN_1 => "DB426_ALARMS_WARNINGS".CLADDING_POWDER_FEEDER."718231",
                           oALARM_DISK_SPEED_BELOW_LOW_LIMIT_LN_1 => "DB426_ALARMS_WARNINGS".CLADDING_POWDER_FEEDER."718232",
                           oALARM_STIRRER_SPEED_BELOW_LOW_LIMIT_LN_1 => "DB426_ALARMS_WARNINGS".CLADDING_POWDER_FEEDER."718233",
                           oALARM_GAS_FLOW_ABOVE_HIGH_LIMIT_LN_1 => "DB426_ALARMS_WARNINGS".CLADDING_POWDER_FEEDER."718234",
                           oALARM_DISK_SPEED_ABOVE_HIGH_LIMIT_LN_1 => "DB426_ALARMS_WARNINGS".CLADDING_POWDER_FEEDER."718235",
                           oALARM_STIRRER_SPEED_ABOVE_HIGH_LIMIT_LN_1 => "DB426_ALARMS_WARNINGS".CLADDING_POWDER_FEEDER."718236",
                           oALARM_CARRIER_GAS_INLET_PRESSURE_TOO_LOW_LN_1 => "DB426_ALARMS_WARNINGS".CLADDING_POWDER_FEEDER."718237",
                           oALARM_DISK_MOTOR_PLUGGED_IN_AND_READY_LN_1 => "DB426_ALARMS_WARNINGS".CLADDING_POWDER_FEEDER."718238",
                           oALARM_STIRRER_PLUGGED_IN_AND_READY_LN_1 => "DB426_ALARMS_WARNINGS".CLADDING_POWDER_FEEDER."718239",
                           oALARM_COMMUNICATION_RUNNING_LN_1 => "DB426_ALARMS_WARNINGS".CLADDING_POWDER_FEEDER."718240",
                           oALARM_FEEDER_NOT_READY_LN_1 => "DB426_ALARMS_WARNINGS".CLADDING_POWDER_FEEDER."718241",
                           oWARNING_GAS_FLOW_UNDER_LIMIT_LN_1 => "DB426_ALARMS_WARNINGS".WARNINGS."729810",
                           oWARNING_DISK_SPEED_UNDER_LIMIT_LN_1 => "DB426_ALARMS_WARNINGS".WARNINGS."729811",
                           oWARNING_STIRRER_SPEED_UNDER_LIMIT_LN_1 => "DB426_ALARMS_WARNINGS".WARNINGS."729812",
                           oWARNING_GAS_FLOW_OVER_LIMIT_LN_1 => "DB426_ALARMS_WARNINGS".WARNINGS."729813",
                           oWARNING_DISK_SPEED_OVER_LIMIT_LN_1 => "DB426_ALARMS_WARNINGS".WARNINGS."729814",
                           oWARNING_STIRRER_SPEED_OVER_LIMIT_LN_1 => "DB426_ALARMS_WARNINGS".WARNINGS."729815",
                           oALARM_POWDER_LINE_2_CLOGGED => "DB426_ALARMS_WARNINGS".CLADDING_POWDER_FEEDER."718260",
                           oALARM_GAS_FLOW_BELOW_LOW_LIMIT_LN_2 => "DB426_ALARMS_WARNINGS".CLADDING_POWDER_FEEDER."718261",
                           oALARM_DISK_SPEED_BELOW_LOW_LIMIT_LN_2 => "DB426_ALARMS_WARNINGS".CLADDING_POWDER_FEEDER."718262",
                           oALARM_STIRRER_SPEED_BELOW_LOW_LIMIT_LN_2 => "DB426_ALARMS_WARNINGS".CLADDING_POWDER_FEEDER."718263",
                           oALARM_GAS_FLOW_ABOVE_HIGH_LIMIT_LN_2 => "DB426_ALARMS_WARNINGS".CLADDING_POWDER_FEEDER."718264",
                           oALARM_DISK_SPEED_ABOVE_HIGH_LIMIT_LN_2 => "DB426_ALARMS_WARNINGS".CLADDING_POWDER_FEEDER."718265",
                           oALARM_STIRRER_SPEED_ABOVE_HIGH_LIMIT_LN_2 => "DB426_ALARMS_WARNINGS".CLADDING_POWDER_FEEDER."718266",
                           oALARM_CARRIER_GAS_INLET_PRESSURE_TOO_LOW_LN_2 => "DB426_ALARMS_WARNINGS".CLADDING_POWDER_FEEDER."718267",
                           oALARM_DISK_MOTOR_PLUGGED_IN_AND_READY_LN_2 => "DB426_ALARMS_WARNINGS".CLADDING_POWDER_FEEDER."718268",
                           oALARM_STIRRER_PLUGGED_IN_AND_READY_LN_2 => "DB426_ALARMS_WARNINGS".CLADDING_POWDER_FEEDER."718269",
                           oALARM_COMMUNICATION_RUNNING_LN_2 => "DB426_ALARMS_WARNINGS".CLADDING_POWDER_FEEDER."718270",
                           oALARM_FEEDER_NOT_READY_LN_2 => "DB426_ALARMS_WARNINGS".CLADDING_POWDER_FEEDER."718271",
                           oWARNING_GAS_FLOW_UNDER_LIMIT_LN_2 => "DB426_ALARMS_WARNINGS".WARNINGS."729830",
                           oWARNING_DISK_SPEED_UNDER_LIMIT_LN_2 => "DB426_ALARMS_WARNINGS".WARNINGS."729831",
                           oWARNING_STIRRER_SPEED_UNDER_LIMIT_LN_2 => "DB426_ALARMS_WARNINGS".WARNINGS."729832",
                           oWARNING_GAS_FLOW_OVER_LIMIT_LN_2 => "DB426_ALARMS_WARNINGS".WARNINGS."729833",
                           oWARNING_DISK_SPEED_OVER_LIMIT_LN_2 => "DB426_ALARMS_WARNINGS".WARNINGS."729834",
                           oWARNING_STIRRER_SPEED_OVER_LIMIT_LN_2 => "DB426_ALARMS_WARNINGS".WARNINGS."729835");
END_REGION

REGION Network 5: CALL FB21013 POWDER FEEDER 2 HOPPER UNIT 02
   // 2#0000_0001 OPTIONS 0 BIT 0 LINE 1 ENABLED OPTION
   // 2#0000_0010 OPTIONS 0 BIT 1 LINE 2 ENABLED OPTION
   // 2#0000_0100 OPTIONS 0 BIT 2 SPARE
   // 2#0000_1000 OPTIONS 0 BIT 3 SPARE
   // 2#0001_0000 OPTIONS 0 BIT 4 SPARE
   // 2#0010_0000 OPTIONS 0 BIT 5 SPARE
   // 2#0100_0000 OPTIONS 0 BIT 6 SPARE
   // 2#1000_0000 OPTIONS 0 BIT 7 SPARE
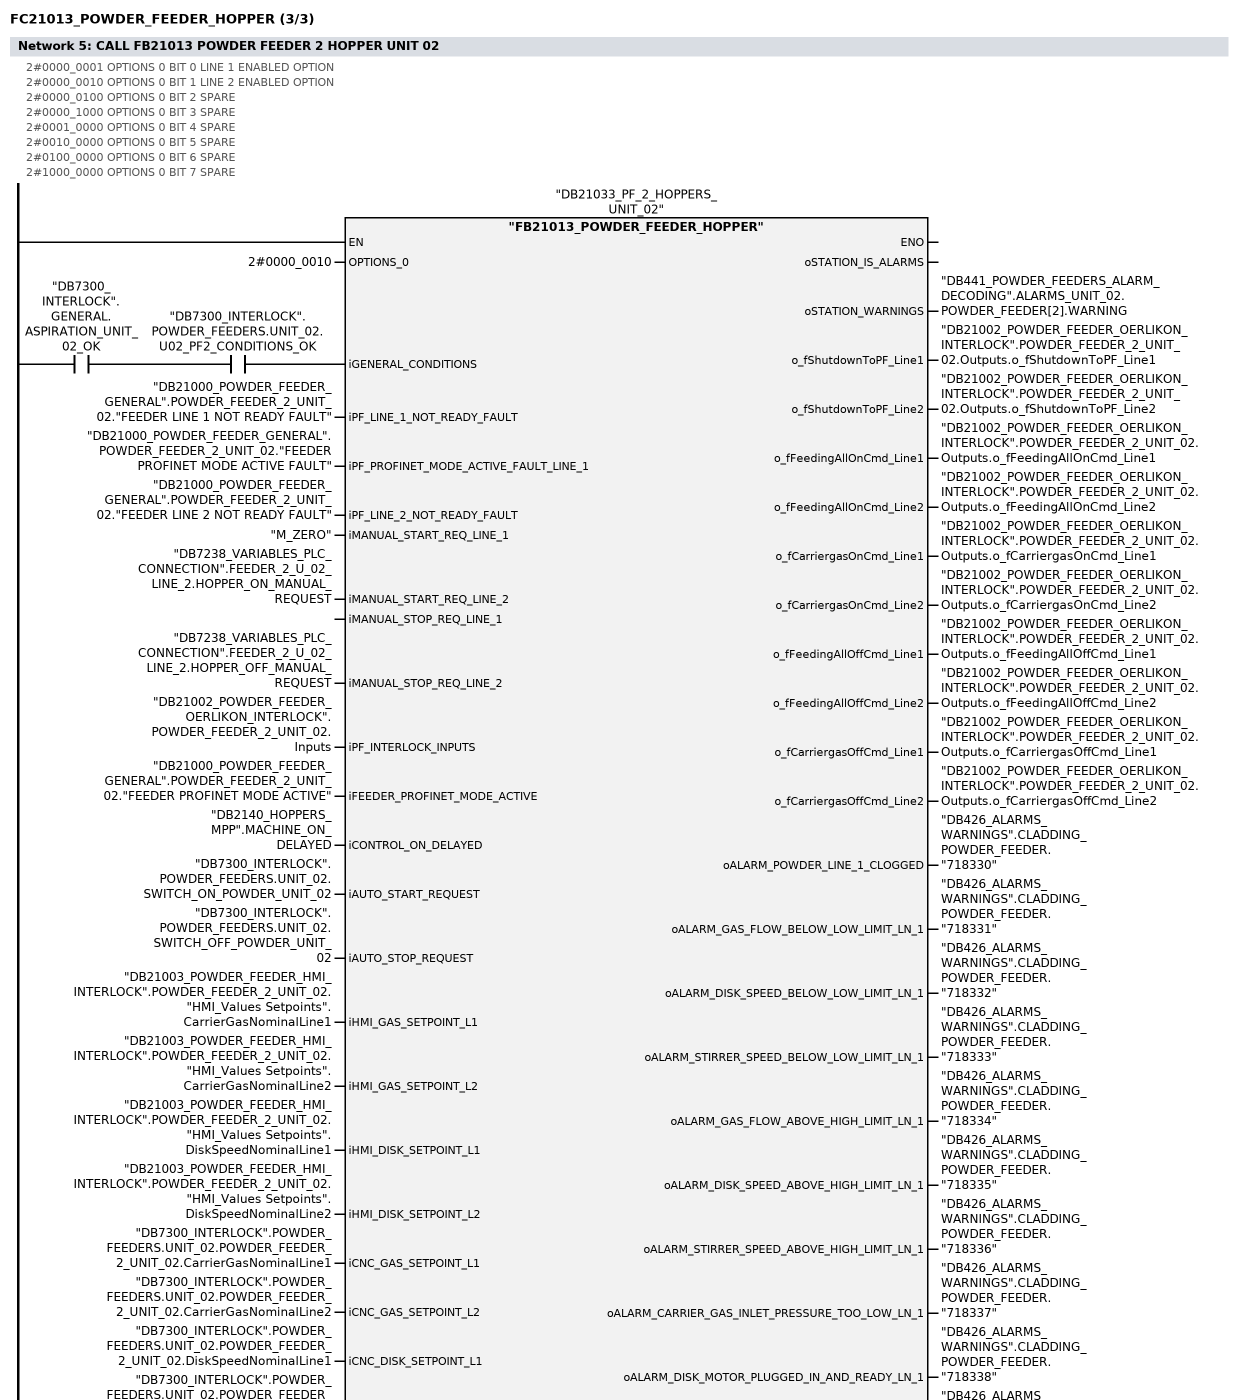
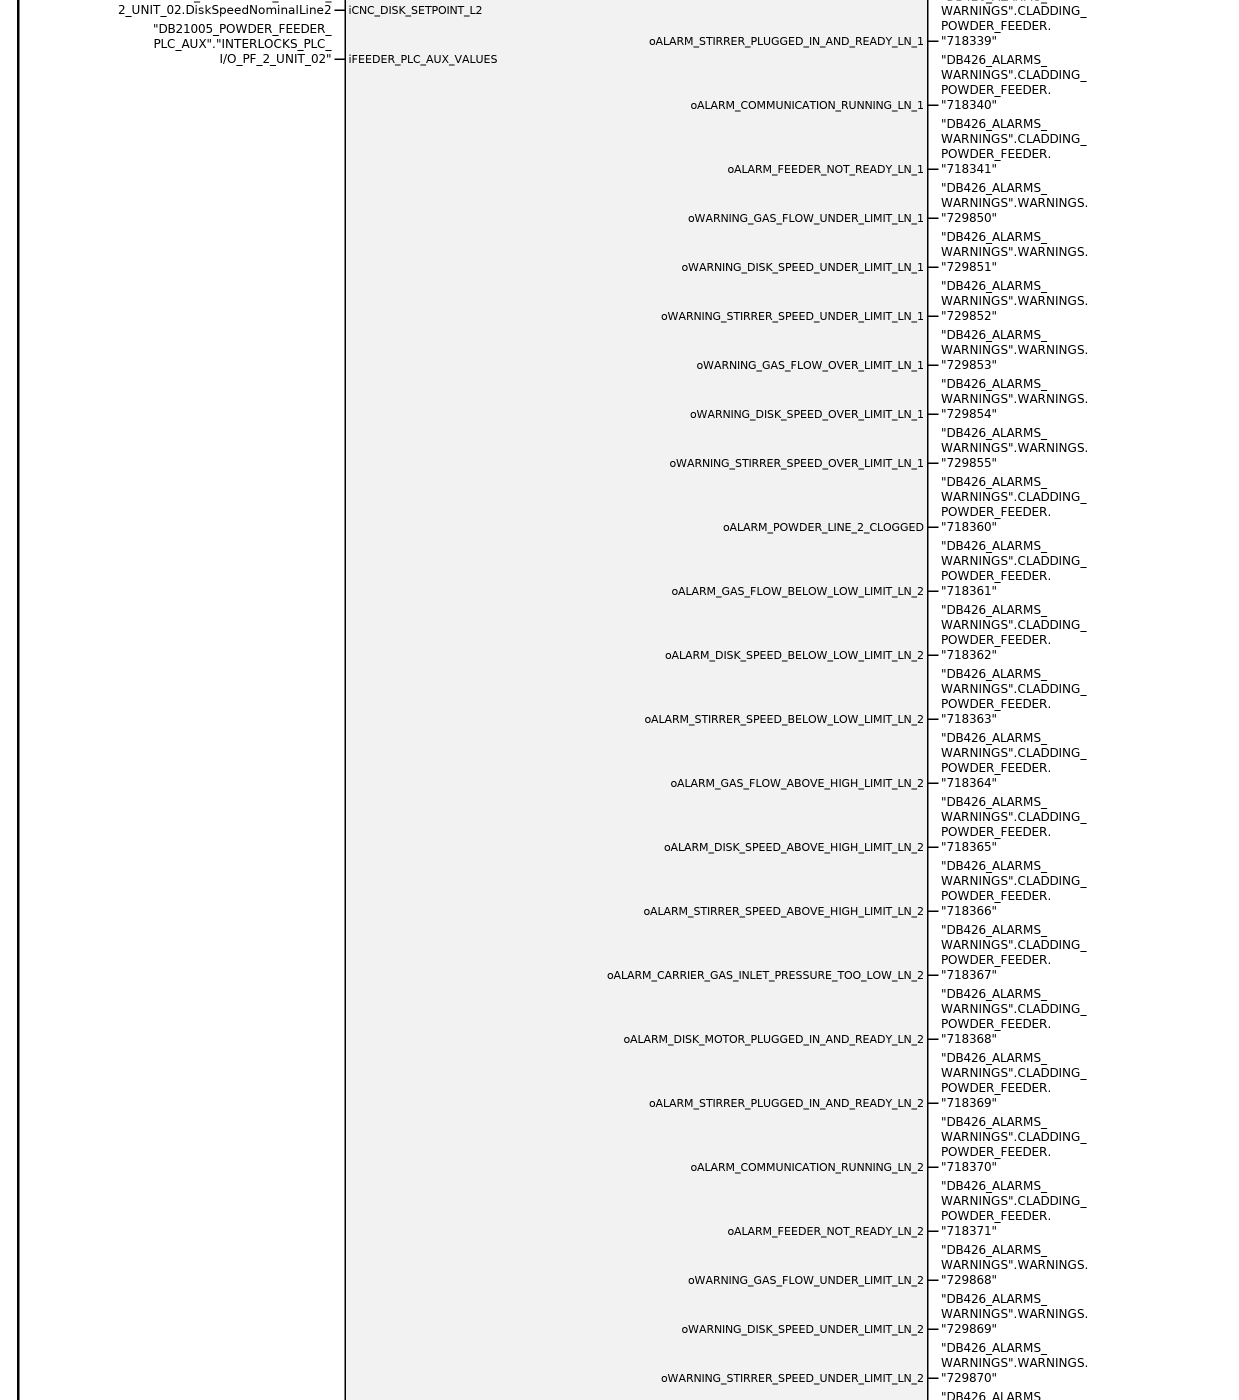
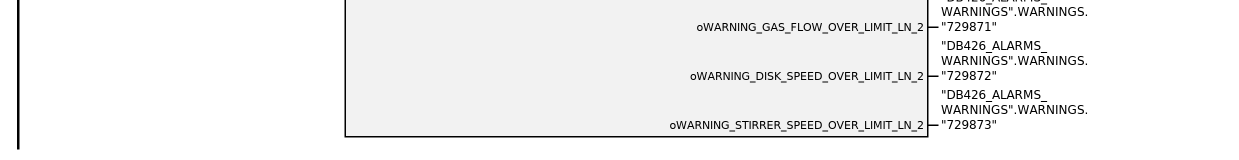
   RUNG wire#powerrail
      "DB21033_PF_2_HOPPERS_UNIT_02"(iGENERAL_CONDITIONS := wire#w1, OPTIONS_0 := 2#0000_0010, iPF_LINE_1_NOT_READY_FAULT := "DB21000_POWDER_FEEDER_GENERAL".POWDER_FEEDER_2_UNIT_02."FEEDER LINE 1 NOT READY FAULT", iPF_PROFINET_MODE_ACTIVE_FAULT_LINE_1 := "DB21000_POWDER_FEEDER_GENERAL".POWDER_FEEDER_2_UNIT_02."FEEDER PROFINET MODE ACTIVE FAULT", iPF_LINE_2_NOT_READY_FAULT := "DB21000_POWDER_FEEDER_GENERAL".POWDER_FEEDER_2_UNIT_02."FEEDER LINE 2 NOT READY FAULT", iMANUAL_START_REQ_LINE_1 := "M_ZERO", iMANUAL_START_REQ_LINE_2 := "DB7238_VARIABLES_PLC_CONNECTION".FEEDER_2_U_02_LINE_2.HOPPER_ON_MANUAL_REQUEST, iMANUAL_STOP_REQ_LINE_1 :=, iMANUAL_STOP_REQ_LINE_2 := "DB7238_VARIABLES_PLC_CONNECTION".FEEDER_2_U_02_LINE_2.HOPPER_OFF_MANUAL_REQUEST, iPF_INTERLOCK_INPUTS := "DB21002_POWDER_FEEDER_OERLIKON_INTERLOCK".POWDER_FEEDER_2_UNIT_02.Inputs, iFEEDER_PROFINET_MODE_ACTIVE := "DB21000_POWDER_FEEDER_GENERAL".POWDER_FEEDER_2_UNIT_02."FEEDER PROFINET MODE ACTIVE", iCONTROL_ON_DELAYED := "DB2140_HOPPERS_MPP".MACHINE_ON_DELAYED, iAUTO_START_REQUEST := "DB7300_INTERLOCK".POWDER_FEEDERS.UNIT_02.SWITCH_ON_POWDER_UNIT_02, iAUTO_STOP_REQUEST := "DB7300_INTERLOCK".POWDER_FEEDERS.UNIT_02.SWITCH_OFF_POWDER_UNIT_02, iHMI_GAS_SETPOINT_L1 := "DB21003_POWDER_FEEDER_HMI_INTERLOCK".POWDER_FEEDER_2_UNIT_02."HMI_Values Setpoints".CarrierGasNominalLine1, iHMI_GAS_SETPOINT_L2 := "DB21003_POWDER_FEEDER_HMI_INTERLOCK".POWDER_FEEDER_2_UNIT_02."HMI_Values Setpoints".CarrierGasNominalLine2, iHMI_DISK_SETPOINT_L1 := "DB21003_POWDER_FEEDER_HMI_INTERLOCK".POWDER_FEEDER_2_UNIT_02."HMI_Values Setpoints".DiskSpeedNominalLine1, iHMI_DISK_SETPOINT_L2 := "DB21003_POWDER_FEEDER_HMI_INTERLOCK".POWDER_FEEDER_2_UNIT_02."HMI_Values Setpoints".DiskSpeedNominalLine2, iCNC_GAS_SETPOINT_L1 := "DB7300_INTERLOCK".POWDER_FEEDERS.UNIT_02.POWDER_FEEDER_2_UNIT_02.CarrierGasNominalLine1, iCNC_GAS_SETPOINT_L2 := "DB7300_INTERLOCK".POWDER_FEEDERS.UNIT_02.POWDER_FEEDER_2_UNIT_02.CarrierGasNominalLine2, iCNC_DISK_SETPOINT_L1 := "DB7300_INTERLOCK".POWDER_FEEDERS.UNIT_02.POWDER_FEEDER_2_UNIT_02.DiskSpeedNominalLine1, iCNC_DISK_SETPOINT_L2 := "DB7300_INTERLOCK".POWDER_FEEDERS.UNIT_02.POWDER_FEEDER_2_UNIT_02.DiskSpeedNominalLine2, iFEEDER_PLC_AUX_VALUES := "DB21005_POWDER_FEEDER_PLC_AUX"."INTERLOCKS_PLC_I/O_PF_2_UNIT_02", oSTATION_IS_ALARMS =>, oSTATION_WARNINGS => "DB441_POWDER_FEEDERS_ALARM_DECODING".ALARMS_UNIT_02.POWDER_FEEDER[2].WARNING, o_fShutdownToPF_Line1 => "DB21002_POWDER_FEEDER_OERLIKON_INTERLOCK".POWDER_FEEDER_2_UNIT_02.Outputs.o_fShutdownToPF_Line1, o_fShutdownToPF_Line2 => "DB21002_POWDER_FEEDER_OERLIKON_INTERLOCK".POWDER_FEEDER_2_UNIT_02.Outputs.o_fShutdownToPF_Line2, o_fFeedingAllOnCmd_Line1 => "DB21002_POWDER_FEEDER_OERLIKON_INTERLOCK".POWDER_FEEDER_2_UNIT_02.Outputs.o_fFeedingAllOnCmd_Line1, o_fFeedingAllOnCmd_Line2 => "DB21002_POWDER_FEEDER_OERLIKON_INTERLOCK".POWDER_FEEDER_2_UNIT_02.Outputs.o_fFeedingAllOnCmd_Line2, o_fCarriergasOnCmd_Line1 => "DB21002_POWDER_FEEDER_OERLIKON_INTERLOCK".POWDER_FEEDER_2_UNIT_02.Outputs.o_fCarriergasOnCmd_Line1, o_fCarriergasOnCmd_Line2 => "DB21002_POWDER_FEEDER_OERLIKON_INTERLOCK".POWDER_FEEDER_2_UNIT_02.Outputs.o_fCarriergasOnCmd_Line2, o_fFeedingAllOffCmd_Line1 => "DB21002_POWDER_FEEDER_OERLIKON_INTERLOCK".POWDER_FEEDER_2_UNIT_02.Outputs.o_fFeedingAllOffCmd_Line1, o_fFeedingAllOffCmd_Line2 => "DB21002_POWDER_FEEDER_OERLIKON_INTERLOCK".POWDER_FEEDER_2_UNIT_02.Outputs.o_fFeedingAllOffCmd_Line2, o_fCarriergasOffCmd_Line1 => "DB21002_POWDER_FEEDER_OERLIKON_INTERLOCK".POWDER_FEEDER_2_UNIT_02.Outputs.o_fCarriergasOffCmd_Line1, o_fCarriergasOffCmd_Line2 => "DB21002_POWDER_FEEDER_OERLIKON_INTERLOCK".POWDER_FEEDER_2_UNIT_02.Outputs.o_fCarriergasOffCmd_Line2, oALARM_POWDER_LINE_1_CLOGGED => "DB426_ALARMS_WARNINGS".CLADDING_POWDER_FEEDER."718330", oALARM_GAS_FLOW_BELOW_LOW_LIMIT_LN_1 => "DB426_ALARMS_WARNINGS".CLADDING_POWDER_FEEDER."718331", oALARM_DISK_SPEED_BELOW_LOW_LIMIT_LN_1 => "DB426_ALARMS_WARNINGS".CLADDING_POWDER_FEEDER."718332", oALARM_STIRRER_SPEED_BELOW_LOW_LIMIT_LN_1 => "DB426_ALARMS_WARNINGS".CLADDING_POWDER_FEEDER."718333", oALARM_GAS_FLOW_ABOVE_HIGH_LIMIT_LN_1 => "DB426_ALARMS_WARNINGS".CLADDING_POWDER_FEEDER."718334", oALARM_DISK_SPEED_ABOVE_HIGH_LIMIT_LN_1 => "DB426_ALARMS_WARNINGS".CLADDING_POWDER_FEEDER."718335", oALARM_STIRRER_SPEED_ABOVE_HIGH_LIMIT_LN_1 => "DB426_ALARMS_WARNINGS".CLADDING_POWDER_FEEDER."718336", oALARM_CARRIER_GAS_INLET_PRESSURE_TOO_LOW_LN_1 => "DB426_ALARMS_WARNINGS".CLADDING_POWDER_FEEDER."718337", oALARM_DISK_MOTOR_PLUGGED_IN_AND_READY_LN_1 => "DB426_ALARMS_WARNINGS".CLADDING_POWDER_FEEDER."718338", oALARM_STIRRER_PLUGGED_IN_AND_READY_LN_1 => "DB426_ALARMS_WARNINGS".CLADDING_POWDER_FEEDER."718339", oALARM_COMMUNICATION_RUNNING_LN_1 => "DB426_ALARMS_WARNINGS".CLADDING_POWDER_FEEDER."718340", oALARM_FEEDER_NOT_READY_LN_1 => "DB426_ALARMS_WARNINGS".CLADDING_POWDER_FEEDER."718341", oWARNING_GAS_FLOW_UNDER_LIMIT_LN_1 => "DB426_ALARMS_WARNINGS".WARNINGS."729850", oWARNING_DISK_SPEED_UNDER_LIMIT_LN_1 => "DB426_ALARMS_WARNINGS".WARNINGS."729851", oWARNING_STIRRER_SPEED_UNDER_LIMIT_LN_1 => "DB426_ALARMS_WARNINGS".WARNINGS."729852", oWARNING_GAS_FLOW_OVER_LIMIT_LN_1 => "DB426_ALARMS_WARNINGS".WARNINGS."729853", oWARNING_DISK_SPEED_OVER_LIMIT_LN_1 => "DB426_ALARMS_WARNINGS".WARNINGS."729854", oWARNING_STIRRER_SPEED_OVER_LIMIT_LN_1 => "DB426_ALARMS_WARNINGS".WARNINGS."729855", oALARM_POWDER_LINE_2_CLOGGED => "DB426_ALARMS_WARNINGS".CLADDING_POWDER_FEEDER."718360", oALARM_GAS_FLOW_BELOW_LOW_LIMIT_LN_2 => "DB426_ALARMS_WARNINGS".CLADDING_POWDER_FEEDER."718361", oALARM_DISK_SPEED_BELOW_LOW_LIMIT_LN_2 => "DB426_ALARMS_WARNINGS".CLADDING_POWDER_FEEDER."718362", oALARM_STIRRER_SPEED_BELOW_LOW_LIMIT_LN_2 => "DB426_ALARMS_WARNINGS".CLADDING_POWDER_FEEDER."718363", oALARM_GAS_FLOW_ABOVE_HIGH_LIMIT_LN_2 => "DB426_ALARMS_WARNINGS".CLADDING_POWDER_FEEDER."718364", oALARM_DISK_SPEED_ABOVE_HIGH_LIMIT_LN_2 => "DB426_ALARMS_WARNINGS".CLADDING_POWDER_FEEDER."718365", oALARM_STIRRER_SPEED_ABOVE_HIGH_LIMIT_LN_2 => "DB426_ALARMS_WARNINGS".CLADDING_POWDER_FEEDER."718366", oALARM_CARRIER_GAS_INLET_PRESSURE_TOO_LOW_LN_2 => "DB426_ALARMS_WARNINGS".CLADDING_POWDER_FEEDER."718367", oALARM_DISK_MOTOR_PLUGGED_IN_AND_READY_LN_2 => "DB426_ALARMS_WARNINGS".CLADDING_POWDER_FEEDER."718368", oALARM_STIRRER_PLUGGED_IN_AND_READY_LN_2 => "DB426_ALARMS_WARNINGS".CLADDING_POWDER_FEEDER."718369", oALARM_COMMUNICATION_RUNNING_LN_2 => "DB426_ALARMS_WARNINGS".CLADDING_POWDER_FEEDER."718370", oALARM_FEEDER_NOT_READY_LN_2 => "DB426_ALARMS_WARNINGS".CLADDING_POWDER_FEEDER."718371", oWARNING_GAS_FLOW_UNDER_LIMIT_LN_2 => "DB426_ALARMS_WARNINGS".WARNINGS."729868", oWARNING_DISK_SPEED_UNDER_LIMIT_LN_2 => "DB426_ALARMS_WARNINGS".WARNINGS."729869", oWARNING_STIRRER_SPEED_UNDER_LIMIT_LN_2 => "DB426_ALARMS_WARNINGS".WARNINGS."729870", oWARNING_GAS_FLOW_OVER_LIMIT_LN_2 => "DB426_ALARMS_WARNINGS".WARNINGS."729871", oWARNING_DISK_SPEED_OVER_LIMIT_LN_2 => "DB426_ALARMS_WARNINGS".WARNINGS."729872", oWARNING_STIRRER_SPEED_OVER_LIMIT_LN_2 => "DB426_ALARMS_WARNINGS".WARNINGS."729873")
   END_RUNG
   RUNG wire#powerrail
      Contact( "DB7300_INTERLOCK".GENERAL.ASPIRATION_UNIT_02_OK )
      Contact( "DB7300_INTERLOCK".POWDER_FEEDERS.UNIT_02.U02_PF2_CONDITIONS_OK )
   END_RUNG wire#w1
   // the same network as SCL:
   "DB21033_PF_2_HOPPERS_UNIT_02"(OPTIONS_0 := 2#0000_0010,   // "FB21013_POWDER_FEEDER_HOPPER"
                           iGENERAL_CONDITIONS := "DB7300_INTERLOCK".GENERAL.ASPIRATION_UNIT_02_OK AND "DB7300_INTERLOCK".POWDER_FEEDERS.UNIT_02.U02_PF2_CONDITIONS_OK,
                           iPF_LINE_1_NOT_READY_FAULT := "DB21000_POWDER_FEEDER_GENERAL".POWDER_FEEDER_2_UNIT_02."FEEDER LINE 1 NOT READY FAULT",
                           iPF_PROFINET_MODE_ACTIVE_FAULT_LINE_1 := "DB21000_POWDER_FEEDER_GENERAL".POWDER_FEEDER_2_UNIT_02."FEEDER PROFINET MODE ACTIVE FAULT",
                           iPF_LINE_2_NOT_READY_FAULT := "DB21000_POWDER_FEEDER_GENERAL".POWDER_FEEDER_2_UNIT_02."FEEDER LINE 2 NOT READY FAULT",
                           iMANUAL_START_REQ_LINE_1 := "M_ZERO",
                           iMANUAL_START_REQ_LINE_2 := "DB7238_VARIABLES_PLC_CONNECTION".FEEDER_2_U_02_LINE_2.HOPPER_ON_MANUAL_REQUEST,
                           iMANUAL_STOP_REQ_LINE_2 := "DB7238_VARIABLES_PLC_CONNECTION".FEEDER_2_U_02_LINE_2.HOPPER_OFF_MANUAL_REQUEST,
                           iPF_INTERLOCK_INPUTS := "DB21002_POWDER_FEEDER_OERLIKON_INTERLOCK".POWDER_FEEDER_2_UNIT_02.Inputs,
                           iFEEDER_PROFINET_MODE_ACTIVE := "DB21000_POWDER_FEEDER_GENERAL".POWDER_FEEDER_2_UNIT_02."FEEDER PROFINET MODE ACTIVE",
                           iCONTROL_ON_DELAYED := "DB2140_HOPPERS_MPP".MACHINE_ON_DELAYED,
                           iAUTO_START_REQUEST := "DB7300_INTERLOCK".POWDER_FEEDERS.UNIT_02.SWITCH_ON_POWDER_UNIT_02,
                           iAUTO_STOP_REQUEST := "DB7300_INTERLOCK".POWDER_FEEDERS.UNIT_02.SWITCH_OFF_POWDER_UNIT_02,
                           iHMI_GAS_SETPOINT_L1 := "DB21003_POWDER_FEEDER_HMI_INTERLOCK".POWDER_FEEDER_2_UNIT_02."HMI_Values Setpoints".CarrierGasNominalLine1,
                           iHMI_GAS_SETPOINT_L2 := "DB21003_POWDER_FEEDER_HMI_INTERLOCK".POWDER_FEEDER_2_UNIT_02."HMI_Values Setpoints".CarrierGasNominalLine2,
                           iHMI_DISK_SETPOINT_L1 := "DB21003_POWDER_FEEDER_HMI_INTERLOCK".POWDER_FEEDER_2_UNIT_02."HMI_Values Setpoints".DiskSpeedNominalLine1,
                           iHMI_DISK_SETPOINT_L2 := "DB21003_POWDER_FEEDER_HMI_INTERLOCK".POWDER_FEEDER_2_UNIT_02."HMI_Values Setpoints".DiskSpeedNominalLine2,
                           iCNC_GAS_SETPOINT_L1 := "DB7300_INTERLOCK".POWDER_FEEDERS.UNIT_02.POWDER_FEEDER_2_UNIT_02.CarrierGasNominalLine1,
                           iCNC_GAS_SETPOINT_L2 := "DB7300_INTERLOCK".POWDER_FEEDERS.UNIT_02.POWDER_FEEDER_2_UNIT_02.CarrierGasNominalLine2,
                           iCNC_DISK_SETPOINT_L1 := "DB7300_INTERLOCK".POWDER_FEEDERS.UNIT_02.POWDER_FEEDER_2_UNIT_02.DiskSpeedNominalLine1,
                           iCNC_DISK_SETPOINT_L2 := "DB7300_INTERLOCK".POWDER_FEEDERS.UNIT_02.POWDER_FEEDER_2_UNIT_02.DiskSpeedNominalLine2,
                           iFEEDER_PLC_AUX_VALUES := "DB21005_POWDER_FEEDER_PLC_AUX"."INTERLOCKS_PLC_I/O_PF_2_UNIT_02",
                           oSTATION_WARNINGS => "DB441_POWDER_FEEDERS_ALARM_DECODING".ALARMS_UNIT_02.POWDER_FEEDER[2].WARNING,
                           o_fShutdownToPF_Line1 => "DB21002_POWDER_FEEDER_OERLIKON_INTERLOCK".POWDER_FEEDER_2_UNIT_02.Outputs.o_fShutdownToPF_Line1,
                           o_fShutdownToPF_Line2 => "DB21002_POWDER_FEEDER_OERLIKON_INTERLOCK".POWDER_FEEDER_2_UNIT_02.Outputs.o_fShutdownToPF_Line2,
                           o_fFeedingAllOnCmd_Line1 => "DB21002_POWDER_FEEDER_OERLIKON_INTERLOCK".POWDER_FEEDER_2_UNIT_02.Outputs.o_fFeedingAllOnCmd_Line1,
                           o_fFeedingAllOnCmd_Line2 => "DB21002_POWDER_FEEDER_OERLIKON_INTERLOCK".POWDER_FEEDER_2_UNIT_02.Outputs.o_fFeedingAllOnCmd_Line2,
                           o_fCarriergasOnCmd_Line1 => "DB21002_POWDER_FEEDER_OERLIKON_INTERLOCK".POWDER_FEEDER_2_UNIT_02.Outputs.o_fCarriergasOnCmd_Line1,
                           o_fCarriergasOnCmd_Line2 => "DB21002_POWDER_FEEDER_OERLIKON_INTERLOCK".POWDER_FEEDER_2_UNIT_02.Outputs.o_fCarriergasOnCmd_Line2,
                           o_fFeedingAllOffCmd_Line1 => "DB21002_POWDER_FEEDER_OERLIKON_INTERLOCK".POWDER_FEEDER_2_UNIT_02.Outputs.o_fFeedingAllOffCmd_Line1,
                           o_fFeedingAllOffCmd_Line2 => "DB21002_POWDER_FEEDER_OERLIKON_INTERLOCK".POWDER_FEEDER_2_UNIT_02.Outputs.o_fFeedingAllOffCmd_Line2,
                           o_fCarriergasOffCmd_Line1 => "DB21002_POWDER_FEEDER_OERLIKON_INTERLOCK".POWDER_FEEDER_2_UNIT_02.Outputs.o_fCarriergasOffCmd_Line1,
                           o_fCarriergasOffCmd_Line2 => "DB21002_POWDER_FEEDER_OERLIKON_INTERLOCK".POWDER_FEEDER_2_UNIT_02.Outputs.o_fCarriergasOffCmd_Line2,
                           oALARM_POWDER_LINE_1_CLOGGED => "DB426_ALARMS_WARNINGS".CLADDING_POWDER_FEEDER."718330",
                           oALARM_GAS_FLOW_BELOW_LOW_LIMIT_LN_1 => "DB426_ALARMS_WARNINGS".CLADDING_POWDER_FEEDER."718331",
                           oALARM_DISK_SPEED_BELOW_LOW_LIMIT_LN_1 => "DB426_ALARMS_WARNINGS".CLADDING_POWDER_FEEDER."718332",
                           oALARM_STIRRER_SPEED_BELOW_LOW_LIMIT_LN_1 => "DB426_ALARMS_WARNINGS".CLADDING_POWDER_FEEDER."718333",
                           oALARM_GAS_FLOW_ABOVE_HIGH_LIMIT_LN_1 => "DB426_ALARMS_WARNINGS".CLADDING_POWDER_FEEDER."718334",
                           oALARM_DISK_SPEED_ABOVE_HIGH_LIMIT_LN_1 => "DB426_ALARMS_WARNINGS".CLADDING_POWDER_FEEDER."718335",
                           oALARM_STIRRER_SPEED_ABOVE_HIGH_LIMIT_LN_1 => "DB426_ALARMS_WARNINGS".CLADDING_POWDER_FEEDER."718336",
                           oALARM_CARRIER_GAS_INLET_PRESSURE_TOO_LOW_LN_1 => "DB426_ALARMS_WARNINGS".CLADDING_POWDER_FEEDER."718337",
                           oALARM_DISK_MOTOR_PLUGGED_IN_AND_READY_LN_1 => "DB426_ALARMS_WARNINGS".CLADDING_POWDER_FEEDER."718338",
                           oALARM_STIRRER_PLUGGED_IN_AND_READY_LN_1 => "DB426_ALARMS_WARNINGS".CLADDING_POWDER_FEEDER."718339",
                           oALARM_COMMUNICATION_RUNNING_LN_1 => "DB426_ALARMS_WARNINGS".CLADDING_POWDER_FEEDER."718340",
                           oALARM_FEEDER_NOT_READY_LN_1 => "DB426_ALARMS_WARNINGS".CLADDING_POWDER_FEEDER."718341",
                           oWARNING_GAS_FLOW_UNDER_LIMIT_LN_1 => "DB426_ALARMS_WARNINGS".WARNINGS."729850",
                           oWARNING_DISK_SPEED_UNDER_LIMIT_LN_1 => "DB426_ALARMS_WARNINGS".WARNINGS."729851",
                           oWARNING_STIRRER_SPEED_UNDER_LIMIT_LN_1 => "DB426_ALARMS_WARNINGS".WARNINGS."729852",
                           oWARNING_GAS_FLOW_OVER_LIMIT_LN_1 => "DB426_ALARMS_WARNINGS".WARNINGS."729853",
                           oWARNING_DISK_SPEED_OVER_LIMIT_LN_1 => "DB426_ALARMS_WARNINGS".WARNINGS."729854",
                           oWARNING_STIRRER_SPEED_OVER_LIMIT_LN_1 => "DB426_ALARMS_WARNINGS".WARNINGS."729855",
                           oALARM_POWDER_LINE_2_CLOGGED => "DB426_ALARMS_WARNINGS".CLADDING_POWDER_FEEDER."718360",
                           oALARM_GAS_FLOW_BELOW_LOW_LIMIT_LN_2 => "DB426_ALARMS_WARNINGS".CLADDING_POWDER_FEEDER."718361",
                           oALARM_DISK_SPEED_BELOW_LOW_LIMIT_LN_2 => "DB426_ALARMS_WARNINGS".CLADDING_POWDER_FEEDER."718362",
                           oALARM_STIRRER_SPEED_BELOW_LOW_LIMIT_LN_2 => "DB426_ALARMS_WARNINGS".CLADDING_POWDER_FEEDER."718363",
                           oALARM_GAS_FLOW_ABOVE_HIGH_LIMIT_LN_2 => "DB426_ALARMS_WARNINGS".CLADDING_POWDER_FEEDER."718364",
                           oALARM_DISK_SPEED_ABOVE_HIGH_LIMIT_LN_2 => "DB426_ALARMS_WARNINGS".CLADDING_POWDER_FEEDER."718365",
                           oALARM_STIRRER_SPEED_ABOVE_HIGH_LIMIT_LN_2 => "DB426_ALARMS_WARNINGS".CLADDING_POWDER_FEEDER."718366",
                           oALARM_CARRIER_GAS_INLET_PRESSURE_TOO_LOW_LN_2 => "DB426_ALARMS_WARNINGS".CLADDING_POWDER_FEEDER."718367",
                           oALARM_DISK_MOTOR_PLUGGED_IN_AND_READY_LN_2 => "DB426_ALARMS_WARNINGS".CLADDING_POWDER_FEEDER."718368",
                           oALARM_STIRRER_PLUGGED_IN_AND_READY_LN_2 => "DB426_ALARMS_WARNINGS".CLADDING_POWDER_FEEDER."718369",
                           oALARM_COMMUNICATION_RUNNING_LN_2 => "DB426_ALARMS_WARNINGS".CLADDING_POWDER_FEEDER."718370",
                           oALARM_FEEDER_NOT_READY_LN_2 => "DB426_ALARMS_WARNINGS".CLADDING_POWDER_FEEDER."718371",
                           oWARNING_GAS_FLOW_UNDER_LIMIT_LN_2 => "DB426_ALARMS_WARNINGS".WARNINGS."729868",
                           oWARNING_DISK_SPEED_UNDER_LIMIT_LN_2 => "DB426_ALARMS_WARNINGS".WARNINGS."729869",
                           oWARNING_STIRRER_SPEED_UNDER_LIMIT_LN_2 => "DB426_ALARMS_WARNINGS".WARNINGS."729870",
                           oWARNING_GAS_FLOW_OVER_LIMIT_LN_2 => "DB426_ALARMS_WARNINGS".WARNINGS."729871",
                           oWARNING_DISK_SPEED_OVER_LIMIT_LN_2 => "DB426_ALARMS_WARNINGS".WARNINGS."729872",
                           oWARNING_STIRRER_SPEED_OVER_LIMIT_LN_2 => "DB426_ALARMS_WARNINGS".WARNINGS."729873");
END_REGION
END_FUNCTION
